// TwinCAT 3 PLC project Untitled1
// ProgramVersion: 3.1.4023.0
// libraries:
//   Tc2_EtherCAT, * (Beckhoff Automation GmbH)
//   Tc2_Standard, * (Beckhoff Automation GmbH)
//   Tc2_System, * (Beckhoff Automation GmbH)
//   Tc3_Module, * (Beckhoff Automation GmbH)
//   VisuDialogs, * (System)
// project tree:
//   DUTs/ DriveReference.TcDUT, Mat3.TcDUT, Motor.TcDUT, TorqueSensor.TcDUT, Vec3.TcDUT
//   / GlobalTextList.TcGTLO, PlcTask.TcTTO, 视图管理器.TcVMO (not stored)
//   GVLs/ GVL.TcGVL
//   POUs/controller/ IntegratedDrive.TcPOU, LegController.TcPOU
//   POUs/GaitPlanner/ BLegSlip.TcPOU, CurlingGait.TcPOU, CurlingGaitFromSlip.TcPOU, CurlingGaitFromStance.TcPOU, GaitPlanner.TcPOU, LiftBodyGait.TcPOU, RcToCurlingFromSlip.TcPOU, RcToSlipFromCurling.TcPOU, RcToStanceFromSlip.TcPOU, RecoverGait.TcPOU, SwingBodyGait.TcPOU, StaticWalkGait.TcPOU, TrotWalk.TcPOU, WalkSlopeGait.TcPOU
//   POUs/HardwareSetup/ MotorDriveSetup.TcPOU, SdoSetup.TcPOU
//   POUs/ MAIN.TcPOU, UIHandler.TcPOU
//   POUs/tools/ AngleCutFun.TcPOU, atan2Fun.TcPOU, CosGenerator.TcPOU, CubicSpline.TcPOU, ElipseInterpolation.TcPOU, GetPivot.TcPOU, HermitInterpolation.TcPOU, LowpassFilter.TcPOU, Min3Value.TcPOU, MinDistanceValue.TcPOU, RotM.TcPOU, SdoWrite.TcPOU
//   POUs/tools/VectorMath/ Atan2.TcPOU, Inv3.TcPOU, MatMulVec.TcPOU, MatTranspose.TcPOU, SetMat3.TcPOU, SetMat7_3.TcPOU, SetVec3.TcPOU, VecAdd.TcPOU, VecCross.TcPOU, VecMulNum.TcPOU, VecNeg.TcPOU, VecNorm.TcPOU, VecNormalize.TcPOU, VecSum.TcPOU
//   VISUs/ AxisControl.TcVIS, ForceControl.TcVIS, Monitor.TcVIS, RobotUI.TcVIS
// real-time tasks:
//   TASK PlcTask: cycle T#1ms, priority 20, ADS port 350
// I/O:
//   DEVICE Device 3 (EtherCAT), AmsNetId 10.0.0.119.4.1
//     Drive 1 (CiA402 Motor Control Device) [SOMANET CiA402 Drive]
//     Drive 2 (CiA402 Motor Control Device) [SOMANET CiA402 Drive]
//     Drive 3 (CiA402 Motor Control Device) [SOMANET CiA402 Drive]
//     Drive 4 (CiA402 Motor Control Device) [SOMANET CiA402 Drive]
//     Drive 5 (CiA402 Motor Control Device) [SOMANET CiA402 Drive]
//     Drive 6 (CiA402 Motor Control Device) [SOMANET CiA402 Drive]
//     Drive 7 (CiA402 Motor Control Device) [SOMANET CiA402 Drive]
//     Drive 8 (CiA402 Motor Control Device) [SOMANET CiA402 Drive]
//     Drive 9 (CiA402 Motor Control Device) [SOMANET CiA402 Drive]
//     Drive 10 (CiA402 Motor Control Device) [SOMANET CiA402 Drive]
//     Drive 11 (CiA402 Motor Control Device) [SOMANET CiA402 Drive]
//     Drive 12 (CiA402 Motor Control Device) [SOMANET CiA402 Drive]
//     Drive 13 (CiA402 Motor Control Device) [SOMANET CiA402 Drive]
//     Drive 14 (CiA402 Motor Control Device) [SOMANET CiA402 Drive]
//     Drive 15 (CiA402 Motor Control Device) [SOMANET CiA402 Drive]
//     Drive 16 (CiA402 Motor Control Device) [SOMANET CiA402 Drive]
//     Drive 17 (CiA402 Motor Control Device) [SOMANET CiA402 Drive]
//     Drive 18 (CiA402 Motor Control Device) [SOMANET CiA402 Drive]
//     Box 19 (TorqueGateway_IMU) [TorqueGateway_IMU]
//     Box 20 (TorqueGateway_IMU) [TorqueGateway_IMU]
//     Box 21 (TorqueGateway_IMU) [TorqueGateway_IMU]
//     Drive 22 (Diamond) [Diamond EtherCAT Drive]
//     Drive 23 (Diamond) [Diamond EtherCAT Drive]
//     Drive 24 (Diamond) [Diamond EtherCAT Drive]
// variable links:
//   Untitled1/Untitled1 Instance <-> Device 3 (EtherCAT)/Box 19 (TorqueGateway_IMU)
//     PlcTask Inputs/GVL.motorDrive[10].trqSensor.trqsensorValue <-> Axis3 process data mapping/ActTrq
//     PlcTask Inputs/GVL.motorDrive[11].trqSensor.trqsensorValue <-> Axis6 process data mapping/ActTrq
//     PlcTask Inputs/GVL.motorDrive[6].trqSensor.trqsensorValue <-> Axis1 process data mapping/ActTrq
//     PlcTask Inputs/GVL.motorDrive[7].trqSensor.trqsensorValue <-> Axis2 process data mapping/ActTrq
//     PlcTask Inputs/GVL.motorDrive[8].trqSensor.trqsensorValue <-> Axis4 process data mapping/ActTrq
//     PlcTask Inputs/GVL.motorDrive[9].trqSensor.trqsensorValue <-> Axis5 process data mapping/ActTrq
//     PlcTask Outputs/GVL.setTrqSensorZero[0] <-> Para process data mapping/Zero
//   Untitled1/Untitled1 Instance <-> Device 3 (EtherCAT)/Box 20 (TorqueGateway_IMU)
//     PlcTask Inputs/GVL.motorDrive[0].trqSensor.trqsensorValue <-> Axis5 process data mapping/ActTrq
//     PlcTask Inputs/GVL.motorDrive[15].trqSensor.trqsensorValue <-> Axis4 process data mapping/ActTrq
//     PlcTask Inputs/GVL.motorDrive[16].trqSensor.trqsensorValue <-> Axis1 process data mapping/ActTrq
//     PlcTask Inputs/GVL.motorDrive[17].trqSensor.trqsensorValue <-> Axis2 process data mapping/ActTrq
//     PlcTask Inputs/GVL.motorDrive[1].trqSensor.trqsensorValue <-> Axis6 process data mapping/ActTrq
//     PlcTask Inputs/GVL.motorDrive[2].trqSensor.trqsensorValue <-> Axis3 process data mapping/ActTrq
//     PlcTask Inputs/GVL.rpy_inpt[0] <-> POSE process data mapping/roll
//     PlcTask Inputs/GVL.rpy_inpt[1] <-> POSE process data mapping/pitch
//     PlcTask Inputs/GVL.rpy_inpt[2] <-> POSE process data mapping/yaw
//     PlcTask Outputs/GVL.setTrqSensorZero[1] <-> Para process data mapping/Zero
//   Untitled1/Untitled1 Instance <-> Device 3 (EtherCAT)/Box 21 (TorqueGateway_IMU)
//     PlcTask Inputs/GVL.motorDrive[12].trqSensor.trqsensorValue <-> Axis3 process data mapping/ActTrq
//     PlcTask Inputs/GVL.motorDrive[13].trqSensor.trqsensorValue <-> Axis6 process data mapping/ActTrq
//     PlcTask Inputs/GVL.motorDrive[14].trqSensor.trqsensorValue <-> Axis5 process data mapping/ActTrq
//     PlcTask Inputs/GVL.motorDrive[3].trqSensor.trqsensorValue <-> Axis4 process data mapping/ActTrq
//     PlcTask Inputs/GVL.motorDrive[4].trqSensor.trqsensorValue <-> Axis2 process data mapping/ActTrq
//     PlcTask Inputs/GVL.motorDrive[5].trqSensor.trqsensorValue <-> Axis1 process data mapping/ActTrq
//     PlcTask Outputs/GVL.setTrqSensorZero[2] <-> Para process data mapping/Zero
//   Untitled1/Untitled1 Instance <-> Device 3 (EtherCAT)/Drive 1 (CiA402 Motor Control Device)
//     PlcTask Inputs/GVL.motorDrive[11].motor.actualPos <-> TxPDO Mapping 1/Position actual value
//     PlcTask Inputs/GVL.motorDrive[11].motor.actualTrq <-> TxPDO Mapping 1/Torque actual value
//     PlcTask Inputs/GVL.motorDrive[11].motor.actualVel <-> TxPDO Mapping 1/Velocity actual value
//     PlcTask Inputs/GVL.motorDrive[11].motor.opModeDisp <-> TxPDO Mapping 1/Modes of operation display
//     PlcTask Inputs/GVL.motorDrive[11].motor.statusWord <-> TxPDO Mapping 1/Statusword
//     PlcTask Outputs/GVL.motorDrive[11].motor.ctrlWord <-> RxPDO Mapping 1/Controlword
//     PlcTask Outputs/GVL.motorDrive[11].motor.opMode <-> RxPDO Mapping 1/Modes of operation
//     PlcTask Outputs/GVL.motorDrive[11].motor.targetPos <-> RxPDO Mapping 1/Target position
//     PlcTask Outputs/GVL.motorDrive[11].motor.targetTrq <-> RxPDO Mapping 1/Target torque
//     PlcTask Outputs/GVL.motorDrive[11].motor.targetVel <-> RxPDO Mapping 1/Target velocity
//   Untitled1/Untitled1 Instance <-> Device 3 (EtherCAT)/Drive 10 (CiA402 Motor Control Device)
//     PlcTask Inputs/GVL.motorDrive[2].motor.actualPos <-> TxPDO Mapping 1/Position actual value
//     PlcTask Inputs/GVL.motorDrive[2].motor.actualTrq <-> TxPDO Mapping 1/Torque actual value
//     PlcTask Inputs/GVL.motorDrive[2].motor.actualVel <-> TxPDO Mapping 1/Velocity actual value
//     PlcTask Inputs/GVL.motorDrive[2].motor.opModeDisp <-> TxPDO Mapping 1/Modes of operation display
//     PlcTask Inputs/GVL.motorDrive[2].motor.statusWord <-> TxPDO Mapping 1/Statusword
//     PlcTask Outputs/GVL.motorDrive[2].motor.ctrlWord <-> RxPDO Mapping 1/Controlword
//     PlcTask Outputs/GVL.motorDrive[2].motor.opMode <-> RxPDO Mapping 1/Modes of operation
//     PlcTask Outputs/GVL.motorDrive[2].motor.targetPos <-> RxPDO Mapping 1/Target position
//     PlcTask Outputs/GVL.motorDrive[2].motor.targetTrq <-> RxPDO Mapping 1/Target torque
//     PlcTask Outputs/GVL.motorDrive[2].motor.targetVel <-> RxPDO Mapping 1/Target velocity
//   Untitled1/Untitled1 Instance <-> Device 3 (EtherCAT)/Drive 11 (CiA402 Motor Control Device)
//     PlcTask Inputs/GVL.motorDrive[1].motor.actualPos <-> TxPDO Mapping 1/Position actual value
//     PlcTask Inputs/GVL.motorDrive[1].motor.actualTrq <-> TxPDO Mapping 1/Torque actual value
//     PlcTask Inputs/GVL.motorDrive[1].motor.actualVel <-> TxPDO Mapping 1/Velocity actual value
//     PlcTask Inputs/GVL.motorDrive[1].motor.opModeDisp <-> TxPDO Mapping 1/Modes of operation display
//     PlcTask Inputs/GVL.motorDrive[1].motor.statusWord <-> TxPDO Mapping 1/Statusword
//     PlcTask Outputs/GVL.motorDrive[1].motor.ctrlWord <-> RxPDO Mapping 1/Controlword
//     PlcTask Outputs/GVL.motorDrive[1].motor.opMode <-> RxPDO Mapping 1/Modes of operation
//     PlcTask Outputs/GVL.motorDrive[1].motor.targetPos <-> RxPDO Mapping 1/Target position
//     PlcTask Outputs/GVL.motorDrive[1].motor.targetTrq <-> RxPDO Mapping 1/Target torque
//     PlcTask Outputs/GVL.motorDrive[1].motor.targetVel <-> RxPDO Mapping 1/Target velocity
//   Untitled1/Untitled1 Instance <-> Device 3 (EtherCAT)/Drive 12 (CiA402 Motor Control Device)
//     PlcTask Inputs/GVL.motorDrive[0].motor.actualPos <-> TxPDO Mapping 1/Position actual value
//     PlcTask Inputs/GVL.motorDrive[0].motor.actualTrq <-> TxPDO Mapping 1/Torque actual value
//     PlcTask Inputs/GVL.motorDrive[0].motor.actualVel <-> TxPDO Mapping 1/Velocity actual value
//     PlcTask Inputs/GVL.motorDrive[0].motor.opModeDisp <-> TxPDO Mapping 1/Modes of operation display
//     PlcTask Inputs/GVL.motorDrive[0].motor.statusWord <-> TxPDO Mapping 1/Statusword
//     PlcTask Outputs/GVL.motorDrive[0].motor.ctrlWord <-> RxPDO Mapping 1/Controlword
//     PlcTask Outputs/GVL.motorDrive[0].motor.opMode <-> RxPDO Mapping 1/Modes of operation
//     PlcTask Outputs/GVL.motorDrive[0].motor.targetPos <-> RxPDO Mapping 1/Target position
//     PlcTask Outputs/GVL.motorDrive[0].motor.targetTrq <-> RxPDO Mapping 1/Target torque
//     PlcTask Outputs/GVL.motorDrive[0].motor.targetVel <-> RxPDO Mapping 1/Target velocity
//   Untitled1/Untitled1 Instance <-> Device 3 (EtherCAT)/Drive 13 (CiA402 Motor Control Device)
//     PlcTask Inputs/GVL.motorDrive[5].motor.actualPos <-> TxPDO Mapping 1/Position actual value
//     PlcTask Inputs/GVL.motorDrive[5].motor.actualTrq <-> TxPDO Mapping 1/Torque actual value
//     PlcTask Inputs/GVL.motorDrive[5].motor.actualVel <-> TxPDO Mapping 1/Velocity actual value
//     PlcTask Inputs/GVL.motorDrive[5].motor.opModeDisp <-> TxPDO Mapping 1/Modes of operation display
//     PlcTask Inputs/GVL.motorDrive[5].motor.statusWord <-> TxPDO Mapping 1/Statusword
//     PlcTask Outputs/GVL.motorDrive[5].motor.ctrlWord <-> RxPDO Mapping 1/Controlword
//     PlcTask Outputs/GVL.motorDrive[5].motor.opMode <-> RxPDO Mapping 1/Modes of operation
//     PlcTask Outputs/GVL.motorDrive[5].motor.targetPos <-> RxPDO Mapping 1/Target position
//     PlcTask Outputs/GVL.motorDrive[5].motor.targetTrq <-> RxPDO Mapping 1/Target torque
//     PlcTask Outputs/GVL.motorDrive[5].motor.targetVel <-> RxPDO Mapping 1/Target velocity
//   Untitled1/Untitled1 Instance <-> Device 3 (EtherCAT)/Drive 14 (CiA402 Motor Control Device)
//     PlcTask Inputs/GVL.motorDrive[4].motor.actualPos <-> TxPDO Mapping 1/Position actual value
//     PlcTask Inputs/GVL.motorDrive[4].motor.actualTrq <-> TxPDO Mapping 1/Torque actual value
//     PlcTask Inputs/GVL.motorDrive[4].motor.actualVel <-> TxPDO Mapping 1/Velocity actual value
//     PlcTask Inputs/GVL.motorDrive[4].motor.opModeDisp <-> TxPDO Mapping 1/Modes of operation display
//     PlcTask Inputs/GVL.motorDrive[4].motor.statusWord <-> TxPDO Mapping 1/Statusword
//     PlcTask Outputs/GVL.motorDrive[4].motor.ctrlWord <-> RxPDO Mapping 1/Controlword
//     PlcTask Outputs/GVL.motorDrive[4].motor.opMode <-> RxPDO Mapping 1/Modes of operation
//     PlcTask Outputs/GVL.motorDrive[4].motor.targetPos <-> RxPDO Mapping 1/Target position
//     PlcTask Outputs/GVL.motorDrive[4].motor.targetTrq <-> RxPDO Mapping 1/Target torque
//     PlcTask Outputs/GVL.motorDrive[4].motor.targetVel <-> RxPDO Mapping 1/Target velocity
//   Untitled1/Untitled1 Instance <-> Device 3 (EtherCAT)/Drive 15 (CiA402 Motor Control Device)
//     PlcTask Inputs/GVL.motorDrive[3].motor.actualPos <-> TxPDO Mapping 1/Position actual value
//     PlcTask Inputs/GVL.motorDrive[3].motor.actualTrq <-> TxPDO Mapping 1/Torque actual value
//     PlcTask Inputs/GVL.motorDrive[3].motor.actualVel <-> TxPDO Mapping 1/Velocity actual value
//     PlcTask Inputs/GVL.motorDrive[3].motor.opModeDisp <-> TxPDO Mapping 1/Modes of operation display
//     PlcTask Inputs/GVL.motorDrive[3].motor.statusWord <-> TxPDO Mapping 1/Statusword
//     PlcTask Outputs/GVL.motorDrive[3].motor.ctrlWord <-> RxPDO Mapping 1/Controlword
//     PlcTask Outputs/GVL.motorDrive[3].motor.opMode <-> RxPDO Mapping 1/Modes of operation
//     PlcTask Outputs/GVL.motorDrive[3].motor.targetPos <-> RxPDO Mapping 1/Target position
//     PlcTask Outputs/GVL.motorDrive[3].motor.targetTrq <-> RxPDO Mapping 1/Target torque
//     PlcTask Outputs/GVL.motorDrive[3].motor.targetVel <-> RxPDO Mapping 1/Target velocity
//   Untitled1/Untitled1 Instance <-> Device 3 (EtherCAT)/Drive 16 (CiA402 Motor Control Device)
//     PlcTask Inputs/GVL.motorDrive[8].motor.actualPos <-> TxPDO Mapping 1/Position actual value
//     PlcTask Inputs/GVL.motorDrive[8].motor.actualTrq <-> TxPDO Mapping 1/Torque actual value
//     PlcTask Inputs/GVL.motorDrive[8].motor.actualVel <-> TxPDO Mapping 1/Velocity actual value
//     PlcTask Inputs/GVL.motorDrive[8].motor.opModeDisp <-> TxPDO Mapping 1/Modes of operation display
//     PlcTask Inputs/GVL.motorDrive[8].motor.statusWord <-> TxPDO Mapping 1/Statusword
//     PlcTask Outputs/GVL.motorDrive[8].motor.ctrlWord <-> RxPDO Mapping 1/Controlword
//     PlcTask Outputs/GVL.motorDrive[8].motor.opMode <-> RxPDO Mapping 1/Modes of operation
//     PlcTask Outputs/GVL.motorDrive[8].motor.targetPos <-> RxPDO Mapping 1/Target position
//     PlcTask Outputs/GVL.motorDrive[8].motor.targetTrq <-> RxPDO Mapping 1/Target torque
//     PlcTask Outputs/GVL.motorDrive[8].motor.targetVel <-> RxPDO Mapping 1/Target velocity
//   Untitled1/Untitled1 Instance <-> Device 3 (EtherCAT)/Drive 17 (CiA402 Motor Control Device)
//     PlcTask Inputs/GVL.motorDrive[7].motor.actualPos <-> TxPDO Mapping 1/Position actual value
//     PlcTask Inputs/GVL.motorDrive[7].motor.actualTrq <-> TxPDO Mapping 1/Torque actual value
//     PlcTask Inputs/GVL.motorDrive[7].motor.actualVel <-> TxPDO Mapping 1/Velocity actual value
//     PlcTask Inputs/GVL.motorDrive[7].motor.opModeDisp <-> TxPDO Mapping 1/Modes of operation display
//     PlcTask Inputs/GVL.motorDrive[7].motor.statusWord <-> TxPDO Mapping 1/Statusword
//     PlcTask Outputs/GVL.motorDrive[7].motor.ctrlWord <-> RxPDO Mapping 1/Controlword
//     PlcTask Outputs/GVL.motorDrive[7].motor.opMode <-> RxPDO Mapping 1/Modes of operation
//     PlcTask Outputs/GVL.motorDrive[7].motor.targetPos <-> RxPDO Mapping 1/Target position
//     PlcTask Outputs/GVL.motorDrive[7].motor.targetTrq <-> RxPDO Mapping 1/Target torque
//     PlcTask Outputs/GVL.motorDrive[7].motor.targetVel <-> RxPDO Mapping 1/Target velocity
//   Untitled1/Untitled1 Instance <-> Device 3 (EtherCAT)/Drive 18 (CiA402 Motor Control Device)
//     PlcTask Inputs/GVL.motorDrive[6].motor.actualPos <-> TxPDO Mapping 1/Position actual value
//     PlcTask Inputs/GVL.motorDrive[6].motor.actualTrq <-> TxPDO Mapping 1/Torque actual value
//     PlcTask Inputs/GVL.motorDrive[6].motor.actualVel <-> TxPDO Mapping 1/Velocity actual value
//     PlcTask Inputs/GVL.motorDrive[6].motor.opModeDisp <-> TxPDO Mapping 1/Modes of operation display
//     PlcTask Inputs/GVL.motorDrive[6].motor.statusWord <-> TxPDO Mapping 1/Statusword
//     PlcTask Outputs/GVL.motorDrive[6].motor.ctrlWord <-> RxPDO Mapping 1/Controlword
//     PlcTask Outputs/GVL.motorDrive[6].motor.opMode <-> RxPDO Mapping 1/Modes of operation
//     PlcTask Outputs/GVL.motorDrive[6].motor.targetPos <-> RxPDO Mapping 1/Target position
//     PlcTask Outputs/GVL.motorDrive[6].motor.targetTrq <-> RxPDO Mapping 1/Target torque
//     PlcTask Outputs/GVL.motorDrive[6].motor.targetVel <-> RxPDO Mapping 1/Target velocity
//   Untitled1/Untitled1 Instance <-> Device 3 (EtherCAT)/Drive 2 (CiA402 Motor Control Device)
//     PlcTask Inputs/GVL.motorDrive[10].motor.actualPos <-> TxPDO Mapping 1/Position actual value
//     PlcTask Inputs/GVL.motorDrive[10].motor.actualTrq <-> TxPDO Mapping 1/Torque actual value
//     PlcTask Inputs/GVL.motorDrive[10].motor.actualVel <-> TxPDO Mapping 1/Velocity actual value
//     PlcTask Inputs/GVL.motorDrive[10].motor.opModeDisp <-> TxPDO Mapping 1/Modes of operation display
//     PlcTask Inputs/GVL.motorDrive[10].motor.statusWord <-> TxPDO Mapping 1/Statusword
//     PlcTask Outputs/GVL.motorDrive[10].motor.ctrlWord <-> RxPDO Mapping 1/Controlword
//     PlcTask Outputs/GVL.motorDrive[10].motor.opMode <-> RxPDO Mapping 1/Modes of operation
//     PlcTask Outputs/GVL.motorDrive[10].motor.targetPos <-> RxPDO Mapping 1/Target position
//     PlcTask Outputs/GVL.motorDrive[10].motor.targetTrq <-> RxPDO Mapping 1/Target torque
//     PlcTask Outputs/GVL.motorDrive[10].motor.targetVel <-> RxPDO Mapping 1/Target velocity
//   Untitled1/Untitled1 Instance <-> Device 3 (EtherCAT)/Drive 22 (Diamond)
//     PlcTask Inputs/GVL.motorDrive[20].motor.actualPos <-> FeedBack process data mapping/Position actual value
//     PlcTask Inputs/GVL.motorDrive[20].motor.actualTrq <-> FeedBack process data mapping/Torque actual value
//     PlcTask Inputs/GVL.motorDrive[20].motor.actualVel <-> FeedBack process data mapping/Velocity actual value
//     PlcTask Inputs/GVL.motorDrive[20].motor.opModeDisp <-> FeedBack process data mapping/Modes of operation display
//     PlcTask Inputs/GVL.motorDrive[20].motor.statusWord <-> FeedBack process data mapping/Statusword
//     PlcTask Outputs/GVL.motorDrive[20].motor.ctrlWord <-> Reference process data mapping/Controlword
//     PlcTask Outputs/GVL.motorDrive[20].motor.opMode <-> Reference process data mapping/Modes of operation
//     PlcTask Outputs/GVL.motorDrive[20].motor.targetPos <-> Reference process data mapping/Target position
//     PlcTask Outputs/GVL.motorDrive[20].motor.targetTrq <-> Reference process data mapping/Target torque
//     PlcTask Outputs/GVL.motorDrive[20].motor.targetVel <-> Reference process data mapping/Target velocity
//   Untitled1/Untitled1 Instance <-> Device 3 (EtherCAT)/Drive 23 (Diamond)
//     PlcTask Inputs/GVL.motorDrive[19].motor.actualPos <-> FeedBack process data mapping/Position actual value
//     PlcTask Inputs/GVL.motorDrive[19].motor.actualTrq <-> FeedBack process data mapping/Torque actual value
//     PlcTask Inputs/GVL.motorDrive[19].motor.actualVel <-> FeedBack process data mapping/Velocity actual value
//     PlcTask Inputs/GVL.motorDrive[19].motor.opModeDisp <-> FeedBack process data mapping/Modes of operation display
//     PlcTask Inputs/GVL.motorDrive[19].motor.statusWord <-> FeedBack process data mapping/Statusword
//     PlcTask Outputs/GVL.motorDrive[19].motor.ctrlWord <-> Reference process data mapping/Controlword
//     PlcTask Outputs/GVL.motorDrive[19].motor.opMode <-> Reference process data mapping/Modes of operation
//     PlcTask Outputs/GVL.motorDrive[19].motor.targetPos <-> Reference process data mapping/Target position
//     PlcTask Outputs/GVL.motorDrive[19].motor.targetTrq <-> Reference process data mapping/Target torque
//     PlcTask Outputs/GVL.motorDrive[19].motor.targetVel <-> Reference process data mapping/Target velocity
//   Untitled1/Untitled1 Instance <-> Device 3 (EtherCAT)/Drive 24 (Diamond)
//     PlcTask Inputs/GVL.motorDrive[18].motor.actualPos <-> FeedBack process data mapping/Position actual value
//     PlcTask Inputs/GVL.motorDrive[18].motor.actualTrq <-> FeedBack process data mapping/Torque actual value
//     PlcTask Inputs/GVL.motorDrive[18].motor.actualVel <-> FeedBack process data mapping/Velocity actual value
//     PlcTask Inputs/GVL.motorDrive[18].motor.opModeDisp <-> FeedBack process data mapping/Modes of operation display
//     PlcTask Inputs/GVL.motorDrive[18].motor.statusWord <-> FeedBack process data mapping/Statusword
//     PlcTask Outputs/GVL.motorDrive[18].motor.ctrlWord <-> Reference process data mapping/Controlword
//     PlcTask Outputs/GVL.motorDrive[18].motor.opMode <-> Reference process data mapping/Modes of operation
//     PlcTask Outputs/GVL.motorDrive[18].motor.targetPos <-> Reference process data mapping/Target position
//     PlcTask Outputs/GVL.motorDrive[18].motor.targetTrq <-> Reference process data mapping/Target torque
//     PlcTask Outputs/GVL.motorDrive[18].motor.targetVel <-> Reference process data mapping/Target velocity
//   Untitled1/Untitled1 Instance <-> Device 3 (EtherCAT)/Drive 3 (CiA402 Motor Control Device)
//     PlcTask Inputs/GVL.motorDrive[9].motor.actualPos <-> TxPDO Mapping 1/Position actual value
//     PlcTask Inputs/GVL.motorDrive[9].motor.actualTrq <-> TxPDO Mapping 1/Torque actual value
//     PlcTask Inputs/GVL.motorDrive[9].motor.actualVel <-> TxPDO Mapping 1/Velocity actual value
//     PlcTask Inputs/GVL.motorDrive[9].motor.opModeDisp <-> TxPDO Mapping 1/Modes of operation display
//     PlcTask Inputs/GVL.motorDrive[9].motor.statusWord <-> TxPDO Mapping 1/Statusword
//     PlcTask Outputs/GVL.motorDrive[9].motor.ctrlWord <-> RxPDO Mapping 1/Controlword
//     PlcTask Outputs/GVL.motorDrive[9].motor.opMode <-> RxPDO Mapping 1/Modes of operation
//     PlcTask Outputs/GVL.motorDrive[9].motor.targetPos <-> RxPDO Mapping 1/Target position
//     PlcTask Outputs/GVL.motorDrive[9].motor.targetTrq <-> RxPDO Mapping 1/Target torque
//     PlcTask Outputs/GVL.motorDrive[9].motor.targetVel <-> RxPDO Mapping 1/Target velocity
//   Untitled1/Untitled1 Instance <-> Device 3 (EtherCAT)/Drive 4 (CiA402 Motor Control Device)
//     PlcTask Inputs/GVL.motorDrive[14].motor.actualPos <-> TxPDO Mapping 1/Position actual value
//     PlcTask Inputs/GVL.motorDrive[14].motor.actualTrq <-> TxPDO Mapping 1/Torque actual value
//     PlcTask Inputs/GVL.motorDrive[14].motor.actualVel <-> TxPDO Mapping 1/Velocity actual value
//     PlcTask Inputs/GVL.motorDrive[14].motor.opModeDisp <-> TxPDO Mapping 1/Modes of operation display
//     PlcTask Inputs/GVL.motorDrive[14].motor.statusWord <-> TxPDO Mapping 1/Statusword
//     PlcTask Outputs/GVL.motorDrive[14].motor.ctrlWord <-> RxPDO Mapping 1/Controlword
//     PlcTask Outputs/GVL.motorDrive[14].motor.opMode <-> RxPDO Mapping 1/Modes of operation
//     PlcTask Outputs/GVL.motorDrive[14].motor.targetPos <-> RxPDO Mapping 1/Target position
//     PlcTask Outputs/GVL.motorDrive[14].motor.targetTrq <-> RxPDO Mapping 1/Target torque
//     PlcTask Outputs/GVL.motorDrive[14].motor.targetVel <-> RxPDO Mapping 1/Target velocity
//   Untitled1/Untitled1 Instance <-> Device 3 (EtherCAT)/Drive 5 (CiA402 Motor Control Device)
//     PlcTask Inputs/GVL.motorDrive[13].motor.actualPos <-> TxPDO Mapping 1/Position actual value
//     PlcTask Inputs/GVL.motorDrive[13].motor.actualTrq <-> TxPDO Mapping 1/Torque actual value
//     PlcTask Inputs/GVL.motorDrive[13].motor.actualVel <-> TxPDO Mapping 1/Velocity actual value
//     PlcTask Inputs/GVL.motorDrive[13].motor.opModeDisp <-> TxPDO Mapping 1/Modes of operation display
//     PlcTask Inputs/GVL.motorDrive[13].motor.statusWord <-> TxPDO Mapping 1/Statusword
//     PlcTask Outputs/GVL.motorDrive[13].motor.ctrlWord <-> RxPDO Mapping 1/Controlword
//     PlcTask Outputs/GVL.motorDrive[13].motor.opMode <-> RxPDO Mapping 1/Modes of operation
//     PlcTask Outputs/GVL.motorDrive[13].motor.targetPos <-> RxPDO Mapping 1/Target position
//     PlcTask Outputs/GVL.motorDrive[13].motor.targetTrq <-> RxPDO Mapping 1/Target torque
//     PlcTask Outputs/GVL.motorDrive[13].motor.targetVel <-> RxPDO Mapping 1/Target velocity
//   Untitled1/Untitled1 Instance <-> Device 3 (EtherCAT)/Drive 6 (CiA402 Motor Control Device)
//     PlcTask Inputs/GVL.motorDrive[12].motor.actualPos <-> TxPDO Mapping 1/Position actual value
//     PlcTask Inputs/GVL.motorDrive[12].motor.actualTrq <-> TxPDO Mapping 1/Torque actual value
//     PlcTask Inputs/GVL.motorDrive[12].motor.actualVel <-> TxPDO Mapping 1/Velocity actual value
//     PlcTask Inputs/GVL.motorDrive[12].motor.opModeDisp <-> TxPDO Mapping 1/Modes of operation display
//     PlcTask Inputs/GVL.motorDrive[12].motor.statusWord <-> TxPDO Mapping 1/Statusword
//     PlcTask Outputs/GVL.motorDrive[12].motor.ctrlWord <-> RxPDO Mapping 1/Controlword
//     PlcTask Outputs/GVL.motorDrive[12].motor.opMode <-> RxPDO Mapping 1/Modes of operation
//     PlcTask Outputs/GVL.motorDrive[12].motor.targetPos <-> RxPDO Mapping 1/Target position
//     PlcTask Outputs/GVL.motorDrive[12].motor.targetTrq <-> RxPDO Mapping 1/Target torque
//     PlcTask Outputs/GVL.motorDrive[12].motor.targetVel <-> RxPDO Mapping 1/Target velocity
//   Untitled1/Untitled1 Instance <-> Device 3 (EtherCAT)/Drive 7 (CiA402 Motor Control Device)
//     PlcTask Inputs/GVL.motorDrive[17].motor.actualPos <-> TxPDO Mapping 1/Position actual value
//     PlcTask Inputs/GVL.motorDrive[17].motor.actualTrq <-> TxPDO Mapping 1/Torque actual value
//     PlcTask Inputs/GVL.motorDrive[17].motor.actualVel <-> TxPDO Mapping 1/Velocity actual value
//     PlcTask Inputs/GVL.motorDrive[17].motor.opModeDisp <-> TxPDO Mapping 1/Modes of operation display
//     PlcTask Inputs/GVL.motorDrive[17].motor.statusWord <-> TxPDO Mapping 1/Statusword
//     PlcTask Outputs/GVL.motorDrive[17].motor.ctrlWord <-> RxPDO Mapping 1/Controlword
//     PlcTask Outputs/GVL.motorDrive[17].motor.opMode <-> RxPDO Mapping 1/Modes of operation
//     PlcTask Outputs/GVL.motorDrive[17].motor.targetPos <-> RxPDO Mapping 1/Target position
//     PlcTask Outputs/GVL.motorDrive[17].motor.targetTrq <-> RxPDO Mapping 1/Target torque
//     PlcTask Outputs/GVL.motorDrive[17].motor.targetVel <-> RxPDO Mapping 1/Target velocity
//   Untitled1/Untitled1 Instance <-> Device 3 (EtherCAT)/Drive 8 (CiA402 Motor Control Device)
//     PlcTask Inputs/GVL.motorDrive[15].motor.actualPos <-> TxPDO Mapping 1/Position actual value
//     PlcTask Inputs/GVL.motorDrive[15].motor.actualTrq <-> TxPDO Mapping 1/Torque actual value
//     PlcTask Inputs/GVL.motorDrive[15].motor.actualVel <-> TxPDO Mapping 1/Velocity actual value
//     PlcTask Inputs/GVL.motorDrive[15].motor.opModeDisp <-> TxPDO Mapping 1/Modes of operation display
//     PlcTask Inputs/GVL.motorDrive[15].motor.statusWord <-> TxPDO Mapping 1/Statusword
//     PlcTask Outputs/GVL.motorDrive[15].motor.ctrlWord <-> RxPDO Mapping 1/Controlword
//     PlcTask Outputs/GVL.motorDrive[15].motor.opMode <-> RxPDO Mapping 1/Modes of operation
//     PlcTask Outputs/GVL.motorDrive[15].motor.targetPos <-> RxPDO Mapping 1/Target position
//     PlcTask Outputs/GVL.motorDrive[15].motor.targetTrq <-> RxPDO Mapping 1/Target torque
//     PlcTask Outputs/GVL.motorDrive[15].motor.targetVel <-> RxPDO Mapping 1/Target velocity
//   Untitled1/Untitled1 Instance <-> Device 3 (EtherCAT)/Drive 9 (CiA402 Motor Control Device)
//     PlcTask Inputs/GVL.motorDrive[16].motor.actualPos <-> TxPDO Mapping 1/Position actual value
//     PlcTask Inputs/GVL.motorDrive[16].motor.actualTrq <-> TxPDO Mapping 1/Torque actual value
//     PlcTask Inputs/GVL.motorDrive[16].motor.actualVel <-> TxPDO Mapping 1/Velocity actual value
//     PlcTask Inputs/GVL.motorDrive[16].motor.opModeDisp <-> TxPDO Mapping 1/Modes of operation display
//     PlcTask Inputs/GVL.motorDrive[16].motor.statusWord <-> TxPDO Mapping 1/Statusword
//     PlcTask Outputs/GVL.motorDrive[16].motor.ctrlWord <-> RxPDO Mapping 1/Controlword
//     PlcTask Outputs/GVL.motorDrive[16].motor.opMode <-> RxPDO Mapping 1/Modes of operation
//     PlcTask Outputs/GVL.motorDrive[16].motor.targetPos <-> RxPDO Mapping 1/Target position
//     PlcTask Outputs/GVL.motorDrive[16].motor.targetTrq <-> RxPDO Mapping 1/Target torque
//     PlcTask Outputs/GVL.motorDrive[16].motor.targetVel <-> RxPDO Mapping 1/Target velocity

CONFIGURATION Untitled1
    RESOURCE PLC ON TwinCAT3
        TASK PlcTask(INTERVAL := T#1ms, PRIORITY := 20);
        PROGRAM MAIN WITH PlcTask : MAIN;
    END_RESOURCE
END_CONFIGURATION

// ---- DUTs/DriveReference.TcDUT
TYPE DriveReference :
STRUCT
	drive : REFERENCE TO IntegratedDrive;
END_STRUCT
END_TYPE

// ---- DUTs/Mat3.TcDUT
TYPE Mat3 :
STRUCT
	data : ARRAY[0..2, 0..2] OF LREAL;
END_STRUCT
END_TYPE

// ---- DUTs/Motor.TcDUT
TYPE Motor :
STRUCT
	statusWord AT%I*: UINT;
	opModeDisp AT%I*: SINT;
	actualPos  AT%I*: DINT;  
	actualVel  AT%I*: DINT;  
	actualTrq  AT%I*: INT; 
	digInputs  AT%I*: DINT;
	
	ctrlWord   AT%Q*: UINT;
	opMode     AT%Q*: USINT;
    targetPos  AT%Q*: DINT   :=0;  
	targetVel  AT%Q*: DINT   :=0;
	targetTrq  AT%Q*: INT    :=0;
	maxTrq     AT%Q*: INT    :=2000;
END_STRUCT
END_TYPE

// ---- DUTs/TorqueSensor.TcDUT
TYPE TorqueSensor :
STRUCT
	trqsensorValue AT%I* : REAL; 
	targetTrqValue AT%I* : REAL;
    
	actPos         AT%Q* : REAL;
	actVel         AT%Q* : REAL;
	TgtPos         AT%Q* : REAL;
	TgtVel         AT%Q* : REAL;
	TrqOff         AT%Q* : REAL;
	SetCtrlPrm     AT%Q* : USINT; 
	reqReset      : usint := 0;
	
	signalPosSlope: LREAL := 35;
	signalNegSlope: LREAL := 35;
END_STRUCT
END_TYPE

// ---- DUTs/Vec3.TcDUT
TYPE Vec3 :
STRUCT
	data : ARRAY[0..2] OF LREAL;
END_STRUCT
END_TYPE

// ---- GVLs/GVL.TcGVL
{attribute 'qualified_only'}
VAR_GLOBAL
	
	
	(*yk 适应*)
	motor_count :  INT :=20;
	
	
	(* system parameters *)
	sampleRate              : DINT := 1000;
	//count2radianRatio  : LREAL := 5.9921124526782860535862796464529E-6;  // 2*pi/1048576
	count2radianRatio  : ARRAY[0..20] OF LREAL := [2*pi/1048576.0,2*pi/1048576.0,2*pi/1048576.0,
                                                   2*pi/1048576.0,2*pi/1048576.0,2*pi/1048576.0,
                                                   2*pi/1048576.0,2*pi/1048576.0,2*pi/1048576.0,
                                                   2*pi/1048576.0,2*pi/1048576.0,2*pi/1048576.0,
                                                   2*pi/1048576.0,2*pi/1048576.0,2*pi/1048576.0,
                                                   2*pi/1048576.0,2*pi/1048576.0,2*pi/1048576.0,
                                                   2*pi/4096.0/9.0,2*pi/4096.0/9.0,2*pi/4096.0/9.0];	
	(* hardware instances *)
	motorDrive              : ARRAY[0..20] OF IntegratedDrive;
	setTrqSensorZero AT%Q*  : ARRAY[0..2]  OF USINT;
	setCtrlZero      AT%Q*  : ARRAY[0..2]  OF USINT;
	
	(* sdo defs *)
	sdoSetup                : SdoSetup;
	sdoWriteOnce            : SdoWrite;
	
	(* IMU readings *)
	IMUDATA : ARRAY[1..6] OF LREAL;
	roll, pitch, yaw        : LREAL;
	accx, accy, accz        : LREAL;
	(* RPY angle aligned to model axis *)
	rpy_model               : ARRAY[0..2] OF LREAL;
	rpy_inpt 		   AT%I*: ARRAY[0..2] OF REAL;
	
	(* motor init parameters*)
	motorDirs        : ARRAY[0..20] OF INT := [1, -1, 1, 
                                               1, 1, 1,
                                               1, 1, 1,
                                               -1, -1, 1,
											   -1, -1, 1,
											   -1, 1, 1,-1,-1,1];//curling2
	(*trqSensorDirs    : ARRAY[0..19] OF INT := [1, -1, 1, 
                                               1, 1, 1,
                                               1, 1, 1,
                                               -1, -1, 1,
											   -1, -1, 1,
 											   -1, 1, 1,1,1];*)
	trqSensorDirs    : ARRAY[0..20] OF INT := [1, -1, 1, 
                                               1, 1, 1,
                                               1, 1, 1,
                                               -1, -1, 1,
											   -1, -1, 1,
 											   -1, 1, 1,-1,-1,-1];											   
											   
	// yk 按照小腿、大腿、侧摆角给出
	(*posHomeOffsets   : ARRAY[0..19] OF LREAL:= [5.497-pi, 3.9269, 0, 
                                                3.9269-pi, 5.497, 0,
                                                3.9269-pi, 5.497, -pi/2, 
                                                3.9269-pi, 5.497, pi/2,
							 					3.9269-pi, 5.497, 0, 
                                                5.497-pi, 3.9269, 0,0,0];//home position in model*)
	(*posHomeOffsets   : ARRAY[0..20] OF LREAL:= [316.8582*pi/180+0.0844, 103.423*pi/180+0.0636, 0*pi/180-0.012, 
                                                109.534*pi/180+0.0052, 350.2283*pi/180-0.042, 90*pi/180-0.018,
                                                102.1787*pi/180+0.0218, 322.4662*pi/180-0.0564, 90*pi/180-0.035, 
                                                102.1787*pi/180+0.0018, 322.4662*pi/180-0.0184, -90*pi/180+0.072,
							 					109.534*pi/180+0.0392, 350.2283*pi/180-0.061, -90*pi/180+0.032, 
                                                316.8582*pi/180+0.0954, 103.423*pi/180+0.0646,  0*180/pi-0,
												0,0,0*pi/180];//home position in model obtained by calibration board	*)
	posHomeOffsets   : ARRAY[0..20] OF LREAL:= [316.8582*pi/180+0.0844, 103.423*pi/180+0.0636, 0*pi/180-0.012, 
                                                109.534*pi/180+0.0052, 350.2283*pi/180-0.042, 90*pi/180-0.018,
                                                102.1787*pi/180+0.0218, 322.4662*pi/180-0.0564, 90*pi/180-0.035, 
                                                102.1787*pi/180+0.0018, 322.4662*pi/180-0.0184, -90*pi/180+0.072,
							 					109.534*pi/180+0.0392, 350.2283*pi/180-0.061, -90*pi/180+0.032, 
                                                316.8582*pi/180+0.0954, 103.423*pi/180+0.0646,  0*180/pi-0,
												0,0,0*pi/180];//home position in model obtained by calibration board											
														
	(*motorActualHomePosIncrement:ARRAY[0..20] OF DINT:= [-391364,-52566,310018,
														 -412094,-268692,-444796,	
														 -432711,-284347,268081,
														 343587,27385,507790,
														 -90255,27553,164936,
														 -124974,-465365,520356,
														 0,0,0];//increment at home position in model obtained by calibration board 20220104*)	
	motorActualHomePosIncrement:ARRAY[0..20] OF DINT:= [-391364,-52566,-281217,
														 -412094,-268692,-444796,	
														 -432711,-284347,268081,
														 343587,27385,507790,
														 -90255,27553,164936,
														 -124974,-465365,263290,
														 0,0,0];//increment at home position in model obtained by calibration board 20220104												 
														 
	signalPosSlopes   : ARRAY[0..20] OF LREAL := [65, 65, 65, 
                                               65, 65, 65,
                                               65, 65, 65,
                                               65, 65, 65,
											   65, 65, 65,
											   65, 65, 65,1,1,1];
	signalNegSlopes   : ARRAY[0..20] OF LREAL := [65, 65, 65, 
                                               65, 65, 65,
                                               65, 65, 65,
                                               65, 65, 65,
											   65, 65, 65,
											   65, 65, 65,1,1,1];
	homingVels       : ARRAY[0..20] OF LREAL:= [0.01, 0.01,  0.01, 
                                               0.01, 0.01,  0.01,
                                               0.01, 0.01,  0.01, 
                                               0.01, 0.01,  0.01,
											   0.01, 0.01,  0.01, 
                                               0.01, 0.01,  0.01,0,0,0.01];
	AbsMoveTgtPos  :	ARRAY[0..20] OF LREAL :=[0, 0, 0,
                                                          0, 0, 0,
														  0, 0, 0,
														  0, 0, 0,
														  0, 0, 0,
														  0, 0, 0,
			                                              0, 0, 0];												   
	redcClbConsts    : ARRAY[0..20] OF LREAL:= [0.01, 0.01, 0.01, 
                                                0.01, 0.01, 0.01,
                                                0.01, 0.01, 0.01, 
                                                0.01, 0.01, 0.01,
                                                0.01, 0.01, 0.01, 
                                                0.01, 0.01, 0.01,0,0,0];
	KPP_init    	 : ARRAY[0..20] OF LREAL:= [1250, 1250, 1250, 
                                                1250, 1250, 1250,
                                                1250, 1250, 1250, 
                                                1250, 1250, 1250,
                                                1250, 1250, 1250, 
                                                1250, 1250, 1250,0,0,0];	
	(*KPP_init    	 : ARRAY[0..20] OF LREAL:= [1000, 1000, 1000, 
                                                1000, 1000, 1000,
                                                1000, 1000, 1000, 
                                                1000, 1000, 1000,
                                                1000, 1000, 1000, 
                                                1000, 1000, 1000,0,0,0];	*)	
	KPD_init    	 : ARRAY[0..20] OF LREAL:= [25, 25, 25, 
                                                25, 25, 25,
                                                25, 25, 25, 
                                                25, 25, 25,
                                                25, 25, 25, 
                                                25, 25, 25,0,0,0];									
	(*KPD_init    	 : ARRAY[0..20] OF LREAL:= [10, 10, 10, 
                                                10, 10, 10,
                                                10, 10, 10, 
                                                10, 10, 10,
                                                10, 10, 10, 
                                                10, 10, 10,0,0,0];*)
	KFP_init    	 : ARRAY[0..20] OF LREAL:= [0.5, 0.5, 0.5, 
                                                0.5, 0.5, 0.5,
                                                0.5, 0.5, 0.5, 
                                                0.5, 0.5, 0.5,
                                                0.5, 0.5, 0.5, 
                                                0.5, 0.5, 0.5,0,0,0];
	KFI_init    	 : ARRAY[0..20] OF LREAL:= [0.75, 0.75, 0.75, 
                                                0.75, 0.75, 0.75,
                                                0.75, 0.75, 0.75, 
                                                0.75, 0.75, 0.75,
                                                0.75, 0.75, 0.75, 
                                                0.75, 0.75, 0.75,0,0,0];


													
												
	//yk 小腿、大腿、侧摆顺序给出，	电机实际角度值，只有运动学上角度才使用小腿角度+pi，			
	trqCtrlUpperAngs : ARRAY[0..20] OF LREAL:= [360, 360, 180, 
                                                360, 360, 180,
                                                360, 360, 180, 
                                                360, 360, 180,
                                                360, 360, 180, 
                                                360, 360, 180,180,180,360];
	trqCtrlLowerAngs : ARRAY[0..20] OF LREAL:= [0, 0, -180, 
                                                0, 0, -180,
                                                0, 0, -180, 
                                                0, 0, -180,
                                                0, 0, -180, 
                                                0, 0, -180,-180,-180,0];
	normalAngles   : ARRAY[0..20] OF LREAL:= [5.497, 3.9269, 0, 
                                              3.9269, 5.497, 0,
                                              3.9269, 5.497, 0, 
                                              3.9269, 5.497, 0,
                                              3.9269, 5.497, 0, 
                                              5.497, 3.9269, 0,0,0,0];// yk 小腿电机角度一定要小于大腿电机角度，才能保证平行四边形腿结构
	(* Visulization linked variables *)
	uiHandler             : UIHandler;
	
	(* axis command *)
	opModeCmd: ARRAY[0..20] OF USINT;
	enableCmd: ARRAY[0..20] OF BOOL;
	
	(* leg physical parameter *)
	ShankLength : ARRAY[0..5] OF LREAL:=[0.5,0.28,0.28,0.28,0.28,0.5];//RB,RM,RF,LF,LM,LB
	ThighLength : ARRAY[0..5] OF LREAL:=[0.5,0.3,0.3,0.3,0.3,0.5];//RB,RM,RF,LF,LM,LB
	
	(* model *)
	legCtrl               : ARRAY[0..5] OF LegController;
	sagPlaneOffset	  :ARRAY[0..5] OF LREAL:=[0,0.1246,0.1246,-0.1246,-0.1246,0];
	
	tipActualPos          : ARRAY[0..5,0..2] OF LREAL := [0, 0, 0,
                                                          0, 0, 0,
														  0, 0, 0,
														  0, 0, 0,
														  0, 0, 0,
														  0, 0, 0];
    tipActualVel          : ARRAY[0..5,0..2] OF LREAL := [0, 0, 0,
                                                          0, 0, 0,
														  0, 0, 0,
														  0, 0, 0,
														  0, 0, 0,
														  0, 0, 0];
    tipActualFce          : ARRAY[0..5,0..2] OF LREAL := [0, 0, 0,
                                                          0, 0, 0,
														  0, 0, 0,
														  0, 0, 0,
														  0, 0, 0,
														  0, 0, 0];
	// joint pos, vel and fce after hardware-model mapping
	jntActualPos          : ARRAY[0..5,0..2] OF LREAL := [0, 0, 0,
                                                          0, 0, 0,
														  0, 0, 0,
														  0, 0, 0,
														  0, 0, 0,
														  0, 0, 0];
    jntActualVel          : ARRAY[0..5,0..2] OF LREAL := [0, 0, 0,
                                                          0, 0, 0,
														  0, 0, 0,
														  0, 0, 0,
														  0, 0, 0,
														  0, 0, 0];
    jntActualFce          : ARRAY[0..5,0..2] OF LREAL := [0, 0, 0,
                                                          0, 0, 0,
														  0, 0, 0,
														  0, 0, 0,
														  0, 0, 0,
														  0, 0, 0];
	// yk 参考位置和速度按照单腿运动学侧摆、大腿、小腿（+pi）给出
	jntRefPos             : ARRAY[0..5,0..2] OF LREAL;
	jntRefVel             : ARRAY[0..5,0..2] OF LREAL;
	lastjntRefPos         : ARRAY[0..5,0..2] OF LREAL:=[0,0,0,
														0,0,0,
														0,0,0,
														0,0,0,
														0,0,0,
														0,0,0];
	jntRefVelDif          : ARRAY[0..5,0..2] OF LREAL;
	jntRefFce             : ARRAY[0..5,0..2] OF LREAL;
	jntLastRefPos         : ARRAY[0..5,0..2] OF LREAL;
	
	jntRefPosTuning       : ARRAY[0..5,0..2] OF LREAL;
	jntRefVelTuning       : ARRAY[0..5,0..2] OF LREAL;
	jntRefFceTuning       : ARRAY[0..5,0..2] OF LREAL;
	
	jntRefPosLastPlanning:ARRAY[0..5,0..2] OF LREAL;
	
	(*jntRefPosLastPlanningFirstRc:ARRAY[0..5,0..2] OF LREAL:=[0,188.4468*pi/180,322.1064*pi/180,
											 0,312.3065*pi/180,(219.5084-312.3065)*pi/180,	
											 0,312.3065*pi/180,(219.5084-312.3065)*pi/180,
											 0,312.3065*pi/180,(219.5084-312.3065)*pi/180,
									         0,312.3065*pi/180,(219.5084-312.3065)*pi/180,
											 0,188.4468*pi/180,322.1064*pi/180];*)
											 
	(*jntRefPosLastPlanningFirstRc:ARRAY[0..5,0..2] OF LREAL:=[0,194.9664*pi/180,320.003*pi/180,
											 0,302.7132*pi/180,(230.9946-302.7132)*pi/180,	
											 0,302.7132*pi/180,(230.9946-302.7132)*pi/180,
											 0,302.7132*pi/180,(230.9946-302.7132)*pi/180,
									         0,302.7132*pi/180,(230.9946-302.7132)*pi/180,
											 0,194.9664*pi/180,320.003*pi/180];	*)

	jntRefPosLastPlanningFirstRc:ARRAY[0..5,0..2] OF LREAL:=[0,156.4222*pi/180,269.8005*pi/180,
											 0,320.9331*pi/180,(208.0880-320.9331)*pi/180,	
											 0,187.8384*pi/180,(269.4264-187.8384)*pi/180,
											 0,187.8384*pi/180,(269.4264-187.8384)*pi/180,
									         0,320.9331*pi/180,(208.0880-320.9331)*pi/180,
											 0,156.4222*pi/180,269.8005*pi/180];										 
	
	(* axis control *)
	enablebuttonText      : ARRAY[0..20] OF STRING(20);
	enableButton          : ARRAY[0..20] OF BOOL;//赋值给enableCmd,gvl.motorDrive[i].DriverControl(gvl.opModeCmd[i], gvl.enableCmd[i])控制电机
	startHomeButton       : ARRAY[0..20] OF BOOL;//单轴和批量都可以赋值，批量赋值后需要进入单轴控制函数执行走home
	setInitPositionButton : ARRAY[0..20] OF BOOL;//单轴和批量都可以赋值，批量赋值后需要进入单轴控制函数执行走设置初始值，调用驱动器驱动函数设置当前home值进入驱动器
	jogButton             : ARRAY[0..20] OF BOOL;
	jogStopButton         : ARRAY[0..20] OF BOOL; 
	jogVelocity           : ARRAY[0..20] OF LREAL;
	AbsMoveButton		  : ARRAY[0..20] OF BOOL;
	AbsMoveStopButton	  : ARRAY[0..20] OF BOOL;
	
	setTSRZeroButton      : BOOL  := FALSE;
	groupSelector         : UINT  := 0;//单选对应数组号，为其值
	enableGroupButton     : BOOL  := FALSE;
	disableGroupButton    : BOOL  := FALSE;
	homeGroupButton       : BOOL  := FALSE;
	setPosGroupButton     : BOOL  := FALSE;
	jogGroupButton        : BOOL  := FALSE;
	jogStopGroupButton    : BOOL  := FALSE;
    //jogGroupVelocity      : DINT  := -2000;
	jogGroupVelocity      : lreal  := 0.01;
	
	setGroupImpedButton   : BOOL  := FALSE;
	useHardImpedButton    : BOOL  := FALSE;
	useSoftImpedButton    : BOOL  := FALSE;
	kpGroup               : LREAL := 220;
	kdGroup               : LREAL := 30;
	kpTrqGroup            : LREAL := 0.5;
	kiTrqGroup            : LREAL := 0.75;
	
	activeAxisList        : ARRAY[0..9] OF ARRAY[0..17] OF USINT := 
                              [[1,1,1,1,1,1,1,1,1,1,1,1,1,1,1,1,1,1],
                               [1,0,0,1,0,0,1,0,0,1,0,0,1,0,0,1,0,0],
                               [0,1,0,0,1,0,0,1,0,0,1,0,0,1,0,0,1,0],
                               [0,0,1,0,0,1,0,0,1,0,0,1,0,0,1,0,0,1],
                               [1,1,1,0,0,0,0,0,0,0,0,0,0,0,0,0,0,0],
                               [0,0,0,1,1,1,0,0,0,0,0,0,0,0,0,0,0,0],
                               [0,0,0,0,0,0,1,1,1,0,0,0,0,0,0,0,0,0],
                               [0,0,0,0,0,0,0,0,0,1,1,1,0,0,0,0,0,0],
                               [0,0,0,0,0,0,0,0,0,0,0,0,1,1,1,0,0,0],
                               [0,0,0,0,0,0,0,0,0,0,0,0,0,0,0,1,1,1]]; //yk 控制一起走home的驱动器号
	
	axisForceCtrlButton   : ARRAY[0..17] OF BOOL;//控制力控开始结束
	axisForceCtrlModeInd  : ARRAY[0..17] OF BOOL;//显示是否处于力控状态
	forceCtrlGroupButton     : BOOL := FALSE;//批量控制进入力控模式
	forceCtrlGroupOffButton  : BOOL := FALSE;//批量停止进入力控模式

	(* gait control *)
	startGaitButton: BOOL   := FALSE;
	isInGaitMode  :  BOOL   := FALSE;
	isFinished    :  BOOL   := FALSE;
	gaitPlanner   :  GaitPlanner;
	gaitId        :  UINT   := 0;
	gaitNameLists :  ARRAY[0..11] OF WSTRING(20) := ["Recovery", "Walk_static", "LiftBody", "Swing","CurlingFrStand","CurlingFrSlip","RcToSlipFrCurl","RcToCurFrSlip","RcToStandFrSlip","BLegSlip","TrotWalk","WalkSlope"];
	
	RcGaitId:UINT:=0;
	RcGaitNameLists:ARRAY[0..1] OF WSTRING(20):=["RcWalk","RcCurling"];
	
	(* measurement *)
	trqReadings           : ARRAY[0..17] OF LREAL;
	trqOutputs            : ARRAY[0..17] OF LREAL;
	trqOutputs2           : ARRAY[0..17] OF LREAL;
	jntActCurrentMea      : ARRAY[0..17] OF INT;
	jntActualPosMea       : ARRAY[0..3,0..2] OF REAL := [0, 0, 0,
                                                          0, 0, 0,
														  0, 0, 0,
														  0, 0, 0];

    jntActualFceMea       : ARRAY[0..3,0..2] OF REAL := [0, 0, 0,
                                                          0, 0, 0,
														  0, 0, 0,
														  0, 0, 0];
	
	jntRefPosMea          : ARRAY[0..3,0..2] OF REAL;
	jntRefFceMea          : ARRAY[0..3,0..2] OF REAL;
	
	(* global stop to shutdown all drives *)
	emergencyStop: BOOL := FALSE;//针对力控
	emergencyStopCount: INT := 0;
	
	(* trq sensor board *)
	useParamIndex: USINT;
	requireSet: BOOL := FALSE;
	raiseEdgeCount: INT := -1;
	setBit: USINT;
	
	walk_threshold_value:LREAL:=0.3;
    lift_threshold_value:LREAL:=0.3;
	swing_threshold_value:LREAL:=0.3;
	curling_threshold_value:lreal:=0.3;

	//Rc gait
	setRcRefAngButton:BOOL:=FALSE;
	
	//curling
	taskChooseId:UINT:=0;
	taskChooseList:array [0..1] of wstring(20):=["击打","进营"];
	adjust_angle_degree:LREAL:=0;//degree
	target_vel:LREAL:=2;//m/s
	stone_rot_vel:LREAL:=-60;//rpm
	PushVelocityIn:LREAL:=2.3;
	BPA_adjust_angle_degree:LREAL:=0;//degree
	BPA_adjust_x:LREAL:=-0.1;
	BPA_adjust_y:LREAL:=0;
	BLPA_adjust_distance_desire:ARRAY[0..1,0..2] OF LREAL:=[0,0,0,
															0,0,0];//[0,-0.01,0,0,0.01,0]																												
	curlingPushModel        :  UINT   := 0;
	curlingPushModelList :  ARRAY[0..1] OF WSTRING(20) := ["Push", "noPush"];
	PushFinishDurationTimeIn:LREAL:=1;
	slideTimeIn:LREAL:=0.3;
	ArmRetractControl:BOOL:=FALSE;
	AC_AngleDegIn:LREAL:=-40;
	
	gripBallThighTargetAngle:LREAL:=167.5;
	gripBallShankTargetAngle:LREAL:=171;
	
	//init value
	adjust_angle_degree_init:LREAL:=0;//degree
	target_vel_init:LREAL:=2;//m/s
	stone_rot_vel_init:LREAL:=-60;//rpm
	PushVelocityIn_init:LREAL:=2.3;
	BPA_adjust_angle_degree_init:LREAL:=0;//degree
	BPA_adjust_x_init:LREAL:=-0.1;
	BPA_adjust_y_init:LREAL:=0;
	BLPA_adjust_distance_desire_init:ARRAY[0..1,0..2] OF LREAL:=[0,0,0,
															0,0,0];	
	curlingPushModel_init        :  UINT   := 0;	
	PushFinishDurationTimeIn_init:LREAL:=1;
	slideTimeIn_init:LREAL:=0.3;
	ArmRetractControl_init:BOOL:=FALSE;
	AC_AngleDegIn_init:LREAL:=-40;	

	//BLegSlip
	BLegSlip_trot_vel_desire:LREAL:=0;
	BLegSlip_side_vel_desire:LREAL:=0;
	BLegSlip_turn_rate_desire:LREAL:=0;
	BLegSlip_step:ARRAY [0..2] OF LREAL:=[0.05,0.05,0.05];
	
	//TrotWalk
	TrotWalk_trot_vel_desire:LREAL:=0;
	TrotWalk_side_vel_desire:LREAL:=0;
	TrotWalk_turn_rate_desire:LREAL:=0;
	TrotWalk_step:ARRAY [0..2] OF LREAL:=[0.15,0.15,0.15];	
	period_desire:LREAL:=1.4;
	duty_desire:LREAL:=0.5;
	step_height_desire:LREAL:=0.06;
	
	//liftbody
	RestButton:BOOL:=FALSE;
	WorkButton:BOOL:=FALSE;
	ReduceDistance:LREAL:=-0.08;
	IsRest:BOOL:=FALSE;
	IsRcCurling:BOOL:=FALSE;
	IsPreLiftBody:BOOL:=FALSE;
	IsLiftBody:BOOL:=FALSE;
	RcEndFlagLast:BOOL:=FALSE;
	RcStartFlag:BOOL:=FALSE;
	RcEndFlag:BOOL:=FALSE;
	EnterPreLiftBodyCount:UDINT:=0;
	LiftBodyStartFlag:BOOL:=FALSE;
	LiftBodyEndFlag:BOOL:=FALSE;
	LiftBodyEndFlagLast:BOOL:=FALSE;
	
	IsWork:BOOL:=FALSE;
	
END_VAR

// ---- POUs/MAIN.TcPOU
PROGRAM MAIN
VAR
	i : UINT;
	j : UINT;
	count : UDINT := 0;

	tipPos, tipVel, tipFce : ARRAY[0..2] OF LREAL;
END_VAR

//////////////////////////////////////////////////////
//                                                  //
// Initialization                                   //
//                                                  //
//////////////////////////////////////////////////////
IF count = 0 THEN
	// init visulization parameters
	gvl.uiHandler.Initialize();
	// init message
	
	// init device address
	// with sdo settings
	gvl.sdoSetup.SetSlaveAddr();//yk需要根据控制器网址设置地址
	
	
	// init axes configuration
	// Note: Some parameters are downloaded to sdo
	// thus not all of these parameters are actually used
	FOR i := 0 TO 20 DO
		gvl.motorDrive[i].InitParam(
			// actual motor direction with regards to the model definition, -1 or +1
			motorDirIn      := gvl.motorDirs[i],
			// actual trq sensor direction wrt the model defintion, -1 or +1 
			trqSensorDirIn  := gvl.trqSensorDirs[i],
			// position offset at home ,need calibrate
			posHomeOffsetIn := gvl.posHomeOffsets[i],
			// signal positive slope of the torque sensor raw output to Nm
			signalPosSlope  := gvl.signalPosSlopes[i],
			// signal negative slope of the torque sensor raw output to Nm
			signalNegSlope  := gvl.signalNegSlopes[i],
			// home velocity
			homingVel       := gvl.homingVels[i],
			// constant of the coloumb friction, yk阻抗控制的是减速机输出扭矩，默认0.01Nm是作用在电机轴上。
			redcClbConst    := gvl.redcClbConsts[i] * 50,
			// trq ctrl upper angle, if the motor runs over this angle, it will be powered off 
			trqCtrlUpperAng := gvl.trqCtrlUpperAngs[i]/180.0*pi,
			// trq ctrl lower angle, if the motor runs over this angle, it will be powered off 
			trqCtrlLowerAng := gvl.trqCtrlLowerAngs[i]/180.0*Pi,
			// trq ctrl normal angle//电机实际值
			tgtAngleIn      := gvl.normalAngles[i]/180.0*pi,
			motorActualHomePosIncrementIn:=gvl.motorActualHomePosIncrement[i],
			indexIn:=i,
			kVirtualIn:=gvl.KPP_init[i],
			bVirtualIn:=gvl.KPD_init[i],
			kpTrqLoopIn:=gvl.KFP_init[i],
			kiTrqLoopIn:=gvl.KFI_init[i],
			count2radianRatioIn:=gvl.count2radianRatio[i]
		);
	END_FOR
	
	// configure leg parameters to leg controller
	FOR i := 0 TO 5 DO
		gvl.LegCtrl[i].InitParam(
			// leg id
			id := i,
			// length of shank link
			ShankLengthIn := GVL.ShankLength[i],
			// length of thigh link
			ThighLengthIn := GVL.ThighLength[i],
			// sagital plane offset
			sagPlaneOffsetIn:=gvl.sagPlaneOffset[i]);
	END_FOR
	
	// set RC reference
	gvl.jntRefPosLastPlanning:=gvl.jntRefPosLastPlanningFirstRc;
	
END_IF

//////////////////////////////////////////////////////
//                                                  //
// Cyclic control                                   //
//                                                  //
//////////////////////////////////////////////////////

// add count 
count := count + 1;

// write sdos configurations to devices 
// this command will last until the sdo writing ops finished 
 gvl.sdoSetup.InitSdoConfig();//设定走home模式和home对应0，所以角度换算时需要加入home对应实际运动学值,设置扭矩传感器可以删除

// update device feedbacks
FOR i := 0 TO 20 DO
	gvl.motorDrive[i].StatusDisplay();
	gvl.motorDrive[i].CalculateMotorAngle();
	gvl.motorDrive[i].CalibrateTrqData();
END_FOR

// Axis level 
// Group command handling,批量控制，需调用单轴控制实现
gvl.uiHandler.GroupMotionCmdHandling();
gvl.uiHandler.GroupForceCtrlCmdHandling();
// Axis command handling,单轴运动控制和力控
gvl.uiHandler.AxisMotionCmdHandling();
gvl.uiHandler.AxisForceCtrlCmdHandling();
// TrqSensor command handling,扭矩传感器清零
gvl.uiHandler.TrqSensorCmdHandling();
// gait command handling步态控制
gvl.uiHandler.GaitCtrlCmdHandling();

// receive imu data from ads
(*gvl.accx := gvl.IMUDATA[1];
gvl.accy := gvl.IMUDATA[2];
gvl.accz := gvl.IMUDATA[3];
gvl.roll := gvl.IMUDATA[4];
gvl.pitch := gvl.IMUDATA[5];
gvl.yaw  := gvl.IMUDATA[6];

// update robot states
gvl.rpy_model[0] := gvl.roll/180.0*pi;
gvl.rpy_model[1] := gvl.pitch/180.0*pi;
gvl.rpy_model[2] := gvl.yaw/180.0*pi;*)
gvl.roll := gvl.rpy_inpt[0];
gvl.pitch := gvl.rpy_inpt[1];
gvl.yaw  := gvl.rpy_inpt[2];
gvl.rpy_model[0] := gvl.roll/180.0*pi;
gvl.rpy_model[1] := gvl.pitch/180.0*pi;
gvl.rpy_model[2] := gvl.yaw/180.0*pi;


FOR i := 0 TO 5 DO
	FOR j := 0 TO 2 DO
		gvl.legCtrl[i].UpdateDriveFeedbacks(gvl.motorDrive[i*3 + j], j,i);////yk 调用18次，每次调用写入一次腿运动学参数
	END_FOR
	
	gvl.legCtrl[i].ForwardKinetics(
		motorAngles := gvl.legCtrl[i].motorAnglesIn,
		legIndex:=i,
		tipPosition => tipPos);
		
	gvl.legCtrl[i].TipVelocity(
		motorVel := gvl.legCtrl[i].motorAngVelIn,
		motorAng := gvl.legCtrl[i].motorAnglesIn,
		legIndex:=i,
		tipVel   => tipVel);
		
	gvl.legCtrl[i].TipForce(
		motorTrq := gvl.legCtrl[i].jointTorqueIn,
		motorAng := gvl.legCtrl[i].motorAnglesIn,
		legIndex:=i,
		tipFce   => tipFce);
		
	FOR j := 0 TO 2 DO
		gvl.tipActualPos[i, j] := tipPos[j];
		gvl.tipActualVel[i, j] := tipVel[j];
		gvl.tipActualFce[i, j] := tipFce[j];
		gvl.jntActualPos[i, j] := gvl.legCtrl[i].motorAnglesIn[j];
		gvl.jntActualVel[i, j] := gvl.legCtrl[i].motorAngVelIn[j];
		gvl.jntActualFce[i, j] := gvl.legCtrl[i].jointTorqueIn[j];
		gvl.jntLastRefPos[i, j] := gvl.legCtrl[i].motorRefAnglesIn[j];
	END_FOR
END_FOR

///////////////////////////////////////////////////////
// Gait Control

IF gvl.isInGaitMode THEN
	gvl.gaitPlanner.DoPlanning(isDone => gvl.isFinished); 
	
	IF gvl.isFinished OR gvl.emergencyStop THEN
		gvl.gaitPlanner.FinalizeGaitCmd();
		gvl.isInGaitMode := FALSE;
	END_IF
	
	// Download cmds
	FOR i := 0 TO 5 DO
		// copy cmds to each leg,
		gvl.legCtrl[i].SetReference();
		// map ref pos, vel, and fce to actual joints
		FOR j := 0 TO 2 DO
			gvl.legCtrl[i].DownloadDriveCmds(gvl.motorDrive[i*3 + j], j,i);
		END_FOR
	END_FOR
END_IF

// Drive level control
FOR i := 0 TO 20 DO	
	// Mid level control algorithms
	IF NOT gvl.motorDrive[i].isInForceControl THEN
		IF i=18 OR i=19 OR i=20 THEN
			gvl.opModeCmd[i] := 3;
		ELSE
			gvl.opModeCmd[i] := 9;
		END_IF
		IF i=20 THEN
			IF gvl.motorDrive[i].IsAbsMoveState=TRUE THEN
				gvl.opModeCmd[i] := 1;
			ELSE
				gvl.opModeCmd[i] := 3;				
			END_IF
		END_IF
		
		gvl.motorDrive[i].GoHome(); 
		gvl.motorDrive[i].JogControl();
		gvl.motorDrive[i].AbsMove();
	ELSE
		gvl.opModeCmd[i] := 10;
		gvl.motorDrive[i].ImpedControl(
			desiredTorque := 0,
			isExternalIC := FALSE);//阻抗参数已经通过gvl.legCtrl[i].DownloadDriveCmds(gvl.motorDrive[i*3 + j], j)写入，所以这里参考力为0
		
		//gvl.motorDrive[i].ImpedControl2();
		
		// Convert torque (Nm) to current cmd ( per 1/1000 )
		gvl.motorDrive[i].CalculateCurrentCmd();
	END_IF
	
	// Low level control
	gvl.motorDrive[i].DriverControl(gvl.opModeCmd[i], gvl.enableCmd[i]);
END_FOR


(*
yk 需要根据实际更新
// torque sensor board control
gvl.setCtrlZero[0] := 0;
gvl.setCtrlZero[1] := 0;
FOR i := 0 TO 11 DO
	IF i < 6 THEN
		gvl.setCtrlZero[0] := gvl.setCtrlZero[0] OR SHL(gvl.motorDrive[i].trqSensor.reqReset, 5 - i);
	ELSE
		gvl.setCtrlZero[1] := gvl.setCtrlZero[1] OR SHL(gvl.motorDrive[i].trqSensor.reqReset, i - 6);
	END_IF
END_FOR
*)

// clear emergency stop event
IF gvl.emergencyStop THEN
	// count emergency stop event number
	gvl.emergencyStopCount := gvl.emergencyStopCount+1;
	// clear
	gvl.emergencyStop := FALSE;
END_IF

FOR i:=0 TO 5 DO
	FOR j:=0 TO 2 DO
		gvl.jntRefVelDif[i,j]:=(gvl.jntRefPos[i,j]-gvl.lastjntRefPos[i,j])*DINT_TO_LREAL(gvl.sampleRate);
		gvl.lastjntRefPos[i,j]:=gvl.jntRefPos[i,j];
	END_FOR
END_FOR

IF gvl.setRcRefAngButton=TRUE THEN
	gvl.jntRefPosLastPlanning:=gvl.jntRefPosLastPlanningFirstRc;
	gvl.setRcRefAngButton:=FALSE;
END_IF

IF gvl.RestButton=TRUE AND gvl.WorkButton=FALSE THEN
	gvl.ReduceDistance:=-0.08;
	gvl.IsRest:=TRUE;
	gvl.IsWork:=FALSE;
	gvl.LiftBodyStartFlag:=TRUE;
	gvl.LiftBodyEndFlag:=FALSE;
	gvl.LiftBodyEndFlagLast:=FALSE;
	gvl.RestButton:=FALSE;
END_IF
IF gvl.RestButton=FALSE AND gvl.WorkButton=TRUE THEN
	gvl.ReduceDistance:=0.08;
	gvl.IsWork:=TRUE;
	gvl.IsRest:=FALSE;
	gvl.LiftBodyStartFlag:=TRUE;
	gvl.LiftBodyEndFlag:=FALSE;
	gvl.LiftBodyEndFlagLast:=FALSE;
	gvl.WorkButton:=FALSE;
END_IF

IF gvl.IsRest=TRUE THEN
	IF gvl.LiftBodyStartFlag=TRUE THEN
		gvl.LiftBodyStartFlag:=FALSE;
		gvl.gaitId:=2;
		gvl.IsLiftBody:=TRUE;
		IF gvl.ReduceDistance>0 THEN
			gvl.ReduceDistance:=-gvl.ReduceDistance;
		END_IF
		IF ABS(gvl.ReduceDistance)>=0.15 THEN
			gvl.ReduceDistance:=-0.15;
		END_IF 
		GVL.startGaitButton:=TRUE;
		gvl.LiftBodyStartFlag:=FALSE;
		gvl.LiftBodyEndFlag:=FALSE;
	END_IF
	IF gvl.IsLiftBody:=TRUE AND GVL.isInGaitMode=TRUE THEN
		gvl.LiftBodyEndFlag:= gvl.isFinished;
	END_IF	
	IF gvl.LiftBodyEndFlagLast=FALSE AND gvl.LiftBodyEndFlag=TRUE AND gvl.IsLiftBody=TRUE THEN
		gvl.IsLiftBody:=FALSE;
		gvl.IsRest:=FALSE;
	END_IF
	gvl.LiftBodyEndFlagLast:=gvl.LiftBodyEndFlag;	
END_IF

IF gvl.IsWork=TRUE THEN
	IF gvl.LiftBodyStartFlag=TRUE THEN
		gvl.LiftBodyStartFlag:=FALSE;
		gvl.gaitId:=2;
		gvl.IsLiftBody:=TRUE;
		IF gvl.ReduceDistance<0 THEN
			gvl.ReduceDistance:=-gvl.ReduceDistance;
		END_IF
		IF ABS(gvl.ReduceDistance)>=0.15 THEN
			gvl.ReduceDistance:=0.15;
		END_IF 
		GVL.startGaitButton:=TRUE;
		gvl.LiftBodyStartFlag:=FALSE;
		gvl.LiftBodyEndFlag:=FALSE;
	END_IF
	IF gvl.IsLiftBody:=TRUE AND GVL.isInGaitMode=TRUE THEN
		gvl.LiftBodyEndFlag:= gvl.isFinished;
	END_IF	
	IF gvl.LiftBodyEndFlagLast=FALSE AND gvl.LiftBodyEndFlag=TRUE AND gvl.IsLiftBody=TRUE THEN
		gvl.IsLiftBody:=FALSE;
		gvl.IsWork:=FALSE;
	END_IF
	gvl.LiftBodyEndFlagLast:=gvl.LiftBodyEndFlag;	
END_IF

END_PROGRAM

// ---- POUs/UIHandler.TcPOU
FUNCTION_BLOCK UIHandler
VAR_INPUT
END_VAR
VAR_OUTPUT
END_VAR
VAR
	zeroSetCount : DINT := 500;
END_VAR

METHOD PUBLIC AxisForceCtrlCmdHandling : BOOL
VAR_INPUT
END_VAR

VAR
	i: INT;
END_VAR
// Axis command handling
FOR i := 0 TO 17 DO	
	(*IF gvl.emergencyStop THEN
		gvl.axisForceCtrlButton[i] := FALSE;
	END_IF*)
	
	IF GVL.axisForceCtrlButton[i] THEN
		IF NOT gvl.axisForceCtrlModeInd[i] THEN
			gvl.motorDrive[i].startForceControl();
			IF gvl.motorDrive[i].isInForceControl THEN
				gvl.axisForceCtrlModeInd[i] := TRUE;
			ELSE
				gvl.axisForceCtrlButton[i] := FALSE;
			END_IF
		END_IF
	ELSE
		IF gvl.axisForceCtrlModeInd[i] THEN
			gvl.axisForceCtrlModeInd[i] := FALSE;
			gvl.motorDrive[i].StopForceControl();
		END_IF
	END_IF
	
END_FOR
END_METHOD

METHOD PUBLIC AxisMotionCmdHandling : BOOL
VAR_INPUT
END_VAR

VAR
	i: INT;
END_VAR
// Axis command handling,轴的运动最后都通过主函数调用JogControll函数实现，设置home位置，通过主函数调用电机驱动函数实现
FOR i := 0 TO 20 DO	

	IF GVL.enableButton[i] THEN
		GVL.enablebuttonText[i] :='Power Off';
	ELSE
		GVL.enablebuttonText[i] :='Power On';
	END_IF
	
	IF gvl.setInitPositionButton[i] THEN
		gvl.motorDrive[i].SetInitPosition();
		gvl.setInitPositionButton[i] := FALSE;
	END_IF
	
	IF gvl.startHomeButton[i] THEN
		gvl.motorDrive[i].StartGoHome();
		gvl.startHomeButton[i] := FALSE;
	END_IF
	
	IF gvl.AbsMoveButton[i] THEN
		gvl.motorDrive[i].StartAbsMove(GVL.AbsMoveTgtPos[i]);
		gvl.AbsMoveButton[i] := FALSE;
	END_IF
	
	IF gvl.AbsMoveStopButton[i] THEN
		gvl.motorDrive[i].StopAbsMove();
		gvl.AbsMoveStopButton[i] := FALSE;
	END_IF
	
	IF gvl.jogButton[i] THEN
		gvl.motorDrive[i].StartJog(gvl.jogVelocity[i]);
		gvl.jogButton[i] := FALSE;
	END_IF
	
	IF gvl.jogStopButton[i] THEN
		gvl.motorDrive[i].StopJog();
		gvl.jogStopButton[i] := FALSE;
	END_IF
	
	gvl.enableCmd[i] := GVL.enableButton[i]; 
END_FOR
END_METHOD

METHOD PUBLIC GaitCtrlCmdHandling : BOOL
VAR_INPUT
END_VAR
IF gvl.startGaitButton AND NOT gvl.isInGaitMode THEN
	gvl.gaitPlanner.Initialize();
	gvl.isInGaitMode := TRUE;
	gvl.startGaitButton := FALSE;
	gvl.isFinished := FALSE;
END_IF
END_METHOD

METHOD PUBLIC GroupForceCtrlCmdHandling : BOOL
VAR_INPUT
END_VAR

VAR
	i: INT;
END_VAR
IF gvl.forceCtrlGroupButton THEN
	FOR i:= 0 TO 17 DO
		IF gvl.activeAxisList[gvl.groupSelector][i] = 1 THEN
			gvl.axisForceCtrlButton[i] := TRUE;
		END_IF
	END_FOR
	gvl.forceCtrlGroupButton := FALSE;
END_IF

IF gvl.forceCtrlGroupOffButton THEN
	FOR i:= 0 TO 17 DO
		IF gvl.activeAxisList[gvl.groupSelector][i] = 1 THEN
			gvl.axisForceCtrlButton[i] := FALSE;
		END_IF
	END_FOR
	gvl.forceCtrlGroupOffButton := FALSE;
END_IF

IF gvl.useHardImpedButton THEN
	gvl.kpGroup := 2000;
	gvl.kdGroup := 200;
	gvl.kpTrqGroup := 0;
	gvl.kiTrqGroup := 0;
	gvl.useParamIndex := 1;
	gvl.useHardImpedButton := FALSE;
END_IF

IF gvl.useSoftImpedButton THEN
	gvl.kpGroup := 220;
	gvl.kdGroup := 25;
	gvl.kpTrqGroup := 0.65;
	gvl.kiTrqGroup := 0.5;
	gvl.useParamIndex := 0;
	gvl.useSoftImpedButton := FALSE;
END_IF

IF gvl.setGroupImpedButton THEN
	FOR i:= 0 TO 17 DO
		gvl.motorDrive[i].SetImpedanceParam(gvl.kpGroup, gvl.kdGroup, gvl.kpTrqGroup, gvl.kiTrqGroup);
	END_FOR
	gvl.setGroupImpedButton := FALSE;
END_IF
END_METHOD

METHOD PUBLIC GroupMotionCmdHandling : BOOL
VAR_INPUT
END_VAR
VAR_OUTPUT
END_VAR
VAR
	i: INT;
END_VAR
IF gvl.enableGroupButton THEN
	FOR i:= 0 TO 17 DO
		IF gvl.activeAxisList[gvl.groupSelector][i] = 1 THEN
			gvl.enableButton[i] := TRUE;
		END_IF
	END_FOR
	gvl.enableButton[18] := TRUE;
	gvl.enableButton[19] := TRUE;
	gvl.enableButton[20] := TRUE;
	gvl.enableGroupButton := FALSE;
END_IF

IF gvl.disableGroupButton THEN
	FOR i:= 0 TO 17 DO
		IF gvl.activeAxisList[gvl.groupSelector][i] = 1 THEN
			gvl.enableButton[i] := FALSE;
		END_IF
	END_FOR
	gvl.enableButton[18] := FALSE;
	gvl.enableButton[19] := FALSE;
	gvl.enableButton[20] := FALSE;
	gvl.disableGroupButton := FALSE;
END_IF

IF gvl.homeGroupButton THEN
	FOR i:= 0 TO 17 DO
		IF gvl.activeAxisList[gvl.groupSelector][i] = 1 THEN
			gvl.startHomeButton[i] := TRUE;
		END_IF
	END_FOR
	gvl.homeGroupButton := FALSE;
END_IF

IF gvl.setPosGroupButton THEN
	FOR i:= 0 TO 17 DO
		IF gvl.activeAxisList[gvl.groupSelector][i] = 1 THEN
			gvl.setInitPositionButton[i] := TRUE;
		END_IF
	END_FOR
	gvl.setPosGroupButton := FALSE;
END_IF

IF gvl.jogGroupButton THEN
	FOR i:= 0 TO 17 DO
		IF gvl.activeAxisList[gvl.groupSelector][i] = 1 THEN
			gvl.jogButton[i] := TRUE;
			gvl.jogVelocity[i] := gvl.jogGroupVelocity;
		END_IF
	END_FOR
	gvl.jogGroupButton := FALSE;
END_IF

IF gvl.jogStopGroupButton THEN
	FOR i:= 0 TO 17 DO
		IF gvl.activeAxisList[gvl.groupSelector][i] = 1 THEN
			gvl.jogStopButton[i] := TRUE;
		END_IF
	END_FOR
	gvl.jogStopGroupButton := FALSE;
END_IF
END_METHOD

METHOD PUBLIC Initialize : BOOL
VAR_INPUT
END_VAR

VAR
	i: INT;
END_VAR
FOR i := 0 TO 19 DO
	gvl.enableButton[i] := FALSE;
	gvl.startHomeButton[i] := FALSE;
	gvl.setInitPositionButton[i] := FALSE; //yk 设置home位置,home结束需要点击setposition写入
	gvl.jogButton[i] := FALSE;
	gvl.jogVelocity[i] := 0.05;
	gvl.axisForceCtrlButton[i] := FALSE;  //yk 切换为力控模式
	gvl.axisForceCtrlModeInd[i] := FALSE;//yk 指示灯是否力控
END_FOR
END_METHOD

METHOD PUBLIC TrqSensorCmdHandling : BOOL
VAR_INPUT
END_VAR
// TSR control
IF gvl.setTSRZeroButton THEN
	gvl.setTrqSensorZero[0] := 63;
	gvl.setTrqSensorZero[1] := 63;
	gvl.setTrqSensorZero[2] := 63;
	zeroSetCount := zeroSetCount - 1;
ELSE
	gvl.setTrqSensorZero[0] := 0;
	gvl.setTrqSensorZero[1] := 0;
	gvl.setTrqSensorZero[2] := 0;
	zeroSetCount := 500;
END_IF

//往力传感器发送500次清零，防止丢包
IF zeroSetCount <= 0 THEN
	gvl.setTSRZeroButton := FALSE;
END_IF
END_METHOD

END_FUNCTION_BLOCK

// ---- POUs/GaitPlanner/GaitPlanner.TcPOU
FUNCTION_BLOCK GaitPlanner
VAR_INPUT
END_VAR
VAR_OUTPUT
END_VAR
VAR
	gaitCount : UDINT := 0;
	recoverGaitPlanner : RecoverGait;
	StaticwalkGaitPlanner    : StaticWalkGait;
	liftBodyGaitPlanner    : LiftBodyGait;
	swingBodyGaitPlanner : SwingBodyGait;
	CurlingGaitPlanner :CurlingGait;
	CurlingGaitPlanner2 :CurlingGaitFromStance;
	RcToSlipFromCurlingPlanner:RcToSlipFromCurling;
	BLegSlipPlanner:BLegSlip;
	CurlingGaitFromSlipPlanner:CurlingGaitFromSlip;
	RcToCurlingFromSlipPlanner:RcToCurlingFromSlip;
	RcToStanceFromSlipPlanner:RcToStanceFromSlip;
	TrotWalkPlanner:TrotWalk;
	WalkSlopePlanner : WalkSlopeGait;
	
	
END_VAR

METHOD PUBLIC DoPlanning : BOOL
VAR_INPUT
END_VAR
VAR_OUTPUT
	isDone : BOOL;
END_VAR

VAR
	i: INT;
	j: INT;
END_VAR
IF gvl.gaitId = 0 THEN
	recoverGaitPlanner.DoPlanning(gaitCount);
	isDone := recoverGaitPlanner.isFinished;
	FOR i := 0 TO 5 DO
		FOR j := 0 TO 2 DO
			gvl.jntRefPosTuning[i, j] := recoverGaitPlanner.jointPosTarget[i, j];
			gvl.jntRefVelTuning[i, j] := recoverGaitPlanner.jointVelTarget[i, j];
			gvl.jntRefFceTuning[i, j] := recoverGaitPlanner.jointFceTarget[i, j];
		END_FOR
	END_FOR
ELSIF gvl.gaitId = 1 THEN
	StaticwalkGaitPlanner.DoPlanning(gaitCount);
	isDone := StaticwalkGaitPlanner.isFinished;
	FOR i := 0 TO 5 DO
		FOR j := 0 TO 2 DO
			gvl.jntRefPosTuning[i, j] := StaticwalkGaitPlanner.jointPosTarget[i, j];
			gvl.jntRefVelTuning[i, j] := StaticwalkGaitPlanner.jointVelTarget[i, j];
			gvl.jntRefFceTuning[i, j] := StaticwalkGaitPlanner.jointFceTarget[i, j];
		END_FOR
	END_FOR
ELSIF gvl.gaitId = 2 THEN
	liftBodyGaitPlanner.DoPlanning(count:=gaitCount );
	isDone := liftBodyGaitPlanner.isFinished;
	FOR i := 0 TO 5 DO
		FOR j := 0 TO 2 DO
			gvl.jntRefPosTuning[i, j] := liftBodyGaitPlanner.jointPosTarget[i, j];
			gvl.jntRefVelTuning[i, j] := liftBodyGaitPlanner.jointVelTarget[i, j];
			gvl.jntRefFceTuning[i, j] := liftBodyGaitPlanner.jointFceTarget[i, j];
		END_FOR
	END_FOR	

ELSIF gvl.gaitId = 3 THEN
	swingBodyGaitPlanner.DoPlanning(gaitCount);
	isDone := swingBodyGaitPlanner.isFinished;
	FOR i := 0 TO 5 DO
		FOR j := 0 TO 2 DO
			gvl.jntRefPosTuning[i, j] := swingBodyGaitPlanner.jointPosTarget[i, j];
			gvl.jntRefVelTuning[i, j] := swingBodyGaitPlanner.jointVelTarget[i, j];
			gvl.jntRefFceTuning[i, j] := swingBodyGaitPlanner.jointFceTarget[i, j];
		END_FOR
	END_FOR
ELSIF gvl.gaitId = 4 THEN
	CurlingGaitPlanner2.DoPlanning(gaitCount);
	isDone := CurlingGaitPlanner2.isFinished;
	FOR i := 0 TO 5 DO
		FOR j := 0 TO 2 DO
			gvl.jntRefPosTuning[i, j] := CurlingGaitPlanner2.jointPosTarget[i, j];
			gvl.jntRefVelTuning[i, j] := CurlingGaitPlanner2.jointVelTarget[i, j];
			gvl.jntRefFceTuning[i, j] := CurlingGaitPlanner2.jointFceTarget[i, j];
		END_FOR
	END_FOR
ELSIF gvl.gaitId = 5 THEN
	CurlingGaitFromSlipPlanner.DoPlanning(gaitCount);
	isDone := CurlingGaitFromSlipPlanner.isFinished;
	FOR i := 0 TO 5 DO
		FOR j := 0 TO 2 DO
			gvl.jntRefPosTuning[i, j] := CurlingGaitFromSlipPlanner.jointPosTarget[i, j];
			gvl.jntRefVelTuning[i, j] := CurlingGaitFromSlipPlanner.jointVelTarget[i, j];
			gvl.jntRefFceTuning[i, j] := CurlingGaitFromSlipPlanner.jointFceTarget[i, j];
		END_FOR
	END_FOR
ELSIF gvl.gaitId = 6 THEN
	RcToSlipFromCurlingPlanner.DoPlanning(gaitCount);
	isDone := RcToSlipFromCurlingPlanner.isFinished;
	FOR i := 0 TO 5 DO
		FOR j := 0 TO 2 DO
			gvl.jntRefPosTuning[i, j] := RcToSlipFromCurlingPlanner.jointPosTarget[i, j];
			gvl.jntRefVelTuning[i, j] := RcToSlipFromCurlingPlanner.jointVelTarget[i, j];
			gvl.jntRefFceTuning[i, j] := RcToSlipFromCurlingPlanner.jointFceTarget[i, j];
		END_FOR
	END_FOR
ELSIF gvl.gaitId = 7 THEN
	RcToCurlingFromSlipPlanner.DoPlanning(gaitCount);
	isDone := RcToCurlingFromSlipPlanner.isFinished;
	FOR i := 0 TO 5 DO
		FOR j := 0 TO 2 DO
			gvl.jntRefPosTuning[i, j] := RcToCurlingFromSlipPlanner.jointPosTarget[i, j];
			gvl.jntRefVelTuning[i, j] := RcToCurlingFromSlipPlanner.jointVelTarget[i, j];
			gvl.jntRefFceTuning[i, j] := RcToCurlingFromSlipPlanner.jointFceTarget[i, j];
		END_FOR
	END_FOR
ELSIF gvl.gaitId = 8 THEN
	RcToStanceFromSlipPlanner.DoPlanning(gaitCount);
	isDone := RcToStanceFromSlipPlanner.isFinished;
	FOR i := 0 TO 5 DO
		FOR j := 0 TO 2 DO
			gvl.jntRefPosTuning[i, j] := RcToStanceFromSlipPlanner.jointPosTarget[i, j];
			gvl.jntRefVelTuning[i, j] := RcToStanceFromSlipPlanner.jointVelTarget[i, j];
			gvl.jntRefFceTuning[i, j] := RcToStanceFromSlipPlanner.jointFceTarget[i, j];
		END_FOR
	END_FOR
ELSIF gvl.gaitId = 9 THEN
	BLegSlipPlanner.DoPlanning(gaitCount);
	isDone := BLegSlipPlanner.isFinished;
	FOR i := 0 TO 5 DO
		FOR j := 0 TO 2 DO
			gvl.jntRefPosTuning[i, j] := BLegSlipPlanner.jointPosTarget[i, j];
			gvl.jntRefVelTuning[i, j] := BLegSlipPlanner.jointVelTarget[i, j];
			gvl.jntRefFceTuning[i, j] := BLegSlipPlanner.jointFceTarget[i, j];
		END_FOR
	END_FOR
ELSIF gvl.gaitId = 10 THEN
	TrotWalkPlanner.DoPlanning(gaitCount);
	isDone := TrotWalkPlanner.isFinished;
	FOR i := 0 TO 5 DO
		FOR j := 0 TO 2 DO
			gvl.jntRefPosTuning[i, j] := TrotWalkPlanner.jointPosTarget[i, j];
			gvl.jntRefVelTuning[i, j] := TrotWalkPlanner.jointVelTarget[i, j];
			gvl.jntRefFceTuning[i, j] := TrotWalkPlanner.jointFceTarget[i, j];
		END_FOR
	END_FOR
ELSIF gvl.gaitId = 11 THEN
	WalkSlopePlanner.DoPlanning(gaitCount);
	isDone := WalkSlopePlanner.isFinished;
	FOR i := 0 TO 5 DO
		FOR j := 0 TO 2 DO
			gvl.jntRefPosTuning[i, j] := WalkSlopePlanner.jointPosTarget[i, j];
			gvl.jntRefVelTuning[i, j] := WalkSlopePlanner.jointVelTarget[i, j];
			gvl.jntRefFceTuning[i, j] := WalkSlopePlanner.jointFceTarget[i, j];
		END_FOR
	END_FOR
ELSE
	// no gait selected
	FOR i := 0 TO 5 DO
		FOR j := 0 TO 2 DO
			IF ABS(gvl.jntActualPos[i, j]-gvl.lastjntRefPos[i,j])<0.1 THEN
				gvl.jntRefPosTuning[i, j] :=gvl.lastjntRefPos[i,j];
			ELSE
				gvl.jntRefPosTuning[i, j] := gvl.jntActualPos[i, j];				
			END_IF
			gvl.jntRefVelTuning[i, j] := 0;
			gvl.jntRefFceTuning[i, j] := 0;
		END_FOR
	END_FOR
	isDone := TRUE;
END_IF

//Tuning state 
(*FOR i := 0 TO 5 DO
	FOR j := 0 TO 2 DO
			IF ABS(gvl.jntActualPos[i, j]-gvl.lastjntRefPos[i,j])<0.1 THEN
				gvl.jntRefPos[i, j] :=gvl.lastjntRefPos[i,j];
			ELSE
				gvl.jntRefPos[i, j] := gvl.jntActualPos[i, j];				
			END_IF
		gvl.jntRefVel[i, j] := 0;
		gvl.jntRefFce[i, j] := 0;
	END_FOR
END_FOR*)

//Actual employment
gvl.jntRefPos:=gvl.jntRefPosTuning;
gvl.jntRefVel:=gvl.jntRefVelTuning;
gvl.jntRefFce:=gvl.jntRefFceTuning;

gaitCount := gaitCount + 1;
END_METHOD

METHOD PUBLIC FinalizeGaitCmd : BOOL
VAR_INPUT
END_VAR

VAR
	i: INT;
	j: INT;
END_VAR
FOR i := 0 TO 5 DO
	FOR j := 0 TO 2 DO
		//gvl.jntRefPos[i, j] := gvl.jntActualPos[i, j];
		gvl.jntRefVel[i, j] := 0;
		gvl.jntRefFce[i, j] := 0;
	END_FOR
END_FOR
END_METHOD

METHOD PUBLIC Initialize : BOOL
VAR_INPUT
END_VAR
gaitCount := 0;
END_METHOD

END_FUNCTION_BLOCK

// ---- POUs/GaitPlanner/RecoverGait.TcPOU
FUNCTION_BLOCK RecoverGait
VAR_INPUT
END_VAR
VAR_OUTPUT
END_VAR
VAR
	isFinished : BOOL := FALSE;
	tRetract   : LREAL := 3;
	tWait      : LREAL := 1;
	tExtend    : LREAL := 3;
	jntAngStart:ARRAY[0..5,0..2] OF LREAL;
	jntAngRetract0:ARRAY[0..5,0..2] OF LREAL:=[0,150.7997*pi/180,291.8958*pi/180,
											  0,327.8142*pi/180,(196.8366-327.8142)*pi/180,
											  0,172.5134*pi/180,(269.4767-172.5134)*pi/180,
											  0,172.5134*pi/180,(269.4767-172.5134)*pi/180,
											  0,327.8142*pi/180,(196.8366-327.8142)*pi/180,
											  0,150.7997*pi/180,291.8958*pi/180];//walk
	jntAngRetract1:ARRAY[0..5,0..2] OF LREAL:=[0,163.1808*pi/180,297.208*pi/180,
											  0,322.9120*pi/180,(205.1705-322.9120)*pi/180,
											  0,183.8227*pi/180,(269.8634-183.8227)*pi/180,
											  0,183.8227*pi/180,(269.8634-183.8227)*pi/180,
											  0,322.9120*pi/180,(205.1705-322.9120)*pi/180,
											  0,163.1808*pi/180,297.208*pi/180];//curling	
	jntAngRetract:ARRAY[0..5,0..2] OF LREAL	;								  

	jntAngExtend0:ARRAY[0..5,0..2] OF LREAL:=[0,163.1808*pi/180,297.208*pi/180,
											 0,320.9331*pi/180,(208.0880-320.9331)*pi/180,	
											 0,187.8384*pi/180,(269.4264-187.8384)*pi/180,
											 0,187.8384*pi/180,(269.4264-187.8384)*pi/180,
									         0,320.9331*pi/180,(208.0880-320.9331)*pi/180,
											 0,163.1808*pi/180,297.208*pi/180];//walk
	jntAngExtend1:ARRAY[0..5,0..2] OF LREAL:=[0,181.9845*pi/180,299.9603*pi/180,
											 0,302.7132*pi/180,(230.9946-302.7132)*pi/180,	
											 0,222.0252*pi/180,(254.0072-222.0252)*pi/180,
											 0,222.0252*pi/180,(254.0072-222.0252)*pi/180,
									         0,302.7132*pi/180,(230.9946-302.7132)*pi/180,
											 0,181.9845*pi/180,299.9603*pi/180];//curling
	jntAngExtend:ARRAY[0..5,0..2] OF LREAL;										 
											 
										 
	pivot, pivotDot : LREAL;
	getPivot  : GetPivot;	
	fbGetPivot  : GetPivot;
	pvt, pvtDot : LREAL;

	jointPosTarget  : ARRAY[0..5, 0..2] OF LREAL; 
	jointVelTarget  : ARRAY[0..5, 0..2] OF LREAL;  
	jointFceTarget  : ARRAY[0..5, 0..2] OF LREAL;	

	tipForceDesire:ARRAY[0..5,0..2] OF LREAL;
	jntTrqDesire:ARRAY[0..5,0..2] OF LREAL;
	fceLoadTime:LREAL:=0.5;
	tipForceDesireGroupA:ARRAY[0..5,0..2] OF LREAL:=[0,-125,0,
													 0,0,0,
													 0,0,0,
													 0,0,0,
													 0,0,0,
													 0,0,0];
	tipForceDesireGroupB:ARRAY[0..5,0..2] OF LREAL:=[0,0,0,
													 0,0,0,
													 0,0,0,
													 0,0,0,
													 0,0,0,
													 0,-145,0];
	tipForceDesireZeros:ARRAY[0..5,0..2] OF LREAL:=[0,0,0,
													 0,0,0,
													 0,0,0,
													 0,0,0,
													 0,0,0,
													 0,0,0];								 
											 
END_VAR

METHOD PUBLIC DoPlanning : BOOL
VAR_INPUT
		count : UDINT;
END_VAR
VAR
	tTotal: LREAL;
	tNow: LREAL;
	tr:LREAL;
	
	jntPosBegin : ARRAY[0..5, 0..2] OF LREAL;
	jntPosEnd   : ARRAY[0..5, 0..2] OF LREAL;
	
	legExtractRefPosCurling: ARRAY[0..5, 0..2] OF LREAL:=[-0.35,-0.3+0.02,0,
														  0.1,-0.3+0.02,-0.1246,
														  -0.3+0.05,-0.3+0.02,-0.1246,
														  -0.3+0.05,-0.3+0.02,0.1246,
														  0.1,-0.3+0.02,0.1246,
														  -0.35,-0.3+0.02,0];//-0.15 for front leg
	jntExtractRefPosCurling: ARRAY[0..5, 0..2] OF LREAL:=[0,163.1808*pi/180,297.208*pi/180,
											  			  0,322.9120*pi/180,(205.1705-322.9120)*pi/180,
											              0,183.8227*pi/180,(269.8634-183.8227)*pi/180,
											              0,183.8227*pi/180,(269.8634-183.8227)*pi/180,
											              0,322.9120*pi/180,(205.1705-322.9120)*pi/180,
											              0,163.1808*pi/180,297.208*pi/180];
														  
	(*legExtendRefPosCurling: ARRAY[0..5, 0..2] OF LREAL:=[-0.35,-0.3805-0.07,0,
														  0.1,-0.4-0.07,-0.1246,
														  -0.3,-0.4-0.07,-0.1246,
														  -0.3,-0.4-0.07,0.1246,
														  0.1,-0.4-0.07,0.1246,
														  -0.35,-0.3805-0.07,0];//before change tip*)
	legExtendRefPosCurling: ARRAY[0..5, 0..2] OF LREAL:=[-0.35,-0.4-0.07,0,
														  0.1,-0.4-0.07,-0.1246,
														  -0.3+0.05,-0.4-0.07,-0.1246,
														  -0.3+0.05,-0.4-0.07,0.1246,
														  0.1,-0.4-0.07,0.1246,
														  -0.35,-0.4-0.07,0];//-0.15 for front leg														 
	
	jntExtendRefPosCurling: ARRAY[0..5, 0..2] OF LREAL:=[0,181.9845*pi/180,299.9603*pi/180,
											 			 0,302.7132*pi/180,(230.9946-302.7132)*pi/180,	
											             0,222.0252*pi/180,(254.0072-222.0252)*pi/180,
											             0,222.0252*pi/180,(254.0072-222.0252)*pi/180,
									                     0,302.7132*pi/180,(230.9946-302.7132)*pi/180,
											             0,181.9845*pi/180,299.9603*pi/180]	;	
									  
	legExtractRefPosWalk:    ARRAY[0..5, 0..2] OF LREAL:=[-0.35,-0.3+0.08,0,
														  0.1,-0.3209+0.08,-0.1246,
														  -0.3+0.05,-0.3209+0.08,-0.1246,
														  -0.3+0.05,-0.3209+0.08,0.1246,
														  0.1,-0.3209+0.08,0.1246,
														  -0.35,-0.3+0.08,0];	
														  
	jntExtractRefPosWalk: ARRAY[0..5, 0..2] OF LREAL:= [0,150.7997*pi/180,291.8958*pi/180,
											  			0,327.8142*pi/180,(196.8366-327.8142)*pi/180,
											  			0,172.5134*pi/180,(269.4767-172.5134)*pi/180,
											  			0,172.5134*pi/180,(269.4767-172.5134)*pi/180,
											  			0,327.8142*pi/180,(196.8366-327.8142)*pi/180,
											  			0,150.7997*pi/180,291.8958*pi/180];													  
														  
	(*legExtendRefPosWalk: ARRAY[0..5, 0..2] OF LREAL    :=[-0.35,-0.3,0,
														  0.1,-0.3209,-0.1246,
														  -0.3,-0.3209,-0.1246,
														  -0.3,-0.3209,0.1246,
														  0.1,-0.3209,0.1246,
														  -0.35,-0.3,0];//before change tip*)
	legExtendRefPosWalk: ARRAY[0..5, 0..2] OF LREAL    :=[-0.35,-0.3209,0,
														  0.1,-0.3209,-0.1246,
														  -0.3+0.05,-0.3209,-0.1246,
														  -0.3+0.05,-0.3209,0.1246,
														  0.1,-0.3209,0.1246,
														  -0.35,-0.3209,0];														  
														  
														  
	jntExtendRefPosWalk: ARRAY[0..5, 0..2] OF LREAL:=	   [0,163.1808*pi/180,297.208*pi/180,
											 				0,320.9331*pi/180,(208.0880-320.9331)*pi/180,	
											 				0,187.8384*pi/180,(269.4264-187.8384)*pi/180,
															0,187.8384*pi/180,(269.4264-187.8384)*pi/180,
									         				0,320.9331*pi/180,(208.0880-320.9331)*pi/180,
											 				0,163.1808*pi/180,297.208*pi/180];																						 
	i: INT;
	j: INT;
	tempLeg:ARRAY [0..2] OF LREAL;
	tempJnt:ARRAY [0..2] OF LREAL;
	tempRef:ARRAY [0..2] OF LREAL;
	
	tempTipForce:ARRAY [0..2] OF LREAL;
	temJntActPos:ARRAY [0..2] OF LREAL;
	tempDesJntTrq:ARRAY [0..2] OF LREAL;
END_VAR
IF count = 0 THEN
	isFinished := FALSE;
	FOR i:=0 TO 5 DO
		tempLeg[0]:=legExtractRefPosCurling[i,0];tempLeg[1]:=legExtractRefPosCurling[i,1];tempLeg[2]:=legExtractRefPosCurling[i,2];
		tempRef[0]:=jntExtractRefPosCurling[i,0];tempRef[1]:=jntExtractRefPosCurling[i,1];tempRef[2]:=jntExtractRefPosCurling[i,2];
		GVL.legCtrl[i].InverseKinetics(tipPosition:=tempLeg , refPosLast:=tempRef , legIndex:=i , motorAngles=>tempJnt , isSingular=> );
		jntAngRetract1[i,0]:=tempJnt[0];jntAngRetract1[i,1]:=tempJnt[1];jntAngRetract1[i,2]:=tempJnt[2];
		
		tempLeg[0]:=legExtractRefPosWalk[i,0];tempLeg[1]:=legExtractRefPosWalk[i,1];tempLeg[2]:=legExtractRefPosWalk[i,2];
		tempRef[0]:=jntExtractRefPosWalk[i,0];tempRef[1]:=jntExtractRefPosWalk[i,1];tempRef[2]:=jntExtractRefPosWalk[i,2];
		GVL.legCtrl[i].InverseKinetics(tipPosition:=tempLeg , refPosLast:=tempRef , legIndex:=i , motorAngles=>tempJnt , isSingular=> );
		jntAngRetract0[i,0]:=tempJnt[0];jntAngRetract0[i,1]:=tempJnt[1];jntAngRetract0[i,2]:=tempJnt[2];
		
		tempLeg[0]:=legExtendRefPosCurling[i,0];tempLeg[1]:=legExtendRefPosCurling[i,1];tempLeg[2]:=legExtendRefPosCurling[i,2];
		tempRef[0]:=jntExtendRefPosCurling[i,0];tempRef[1]:=jntExtendRefPosCurling[i,1];tempRef[2]:=jntExtendRefPosCurling[i,2];
		GVL.legCtrl[i].InverseKinetics(tipPosition:=tempLeg , refPosLast:=tempRef , legIndex:=i , motorAngles=>tempJnt , isSingular=> );
		jntAngExtend1[i,0]:=tempJnt[0];jntAngExtend1[i,1]:=tempJnt[1];jntAngExtend1[i,2]:=tempJnt[2];		
		
		tempLeg[0]:=legExtendRefPosWalk[i,0];tempLeg[1]:=legExtendRefPosWalk[i,1];tempLeg[2]:=legExtendRefPosWalk[i,2];
		tempRef[0]:=jntExtendRefPosWalk[i,0];tempRef[1]:=jntExtendRefPosWalk[i,1];tempRef[2]:=jntExtendRefPosWalk[i,2];
		GVL.legCtrl[i].InverseKinetics(tipPosition:=tempLeg , refPosLast:=tempRef , legIndex:=i , motorAngles=>tempJnt , isSingular=> );
		jntAngExtend0[i,0]:=tempJnt[0];jntAngExtend0[i,1]:=tempJnt[1];jntAngExtend0[i,2]:=tempJnt[2];		
	END_FOR
	
	IF gvl.RcGaitId=0 THEN
		jntAngRetract:=jntAngRetract0;
		jntAngExtend:=jntAngExtend0;
	ELSE
		jntAngRetract:=jntAngRetract1;
		jntAngExtend:=jntAngExtend1;			
	END_IF
	
	FOR i := 0 TO 5 DO
		FOR j := 0 TO 2 DO
			IF ABS(gvl.jntLastRefPos[i, j] - gvl.jntActualPos[i, j]) < 0.2 THEN
				jntAngStart[i,j] := gvl.jntLastRefPos[i, j];
			ELSE
				jntAngStart[i,j] := gvl.jntActualPos[i, j];
			END_IF
			jntAngStart[i,j]:=MinDistanceValue(jntAngStart[i,j],gvl.jntRefPosLastPlanning[i,j]);
			
		END_FOR
	END_FOR	
	
	tipForceDesire:=tipForceDesireZeros;	
END_IF

IF count<=(tRetract + tWait + tExtend) * gvl.sampleRate THEN //leg 0-2-4 recovery
	
//******************************force compensator******************************
	IF count<=fceLoadTime*gvl.sampleRate THEN
		tr  := UDINT_TO_LREAL(count) / gvl.sampleRate /fceLoadTime;
		fbGetPivot(tNow := tr, tTotal := 1.0, pivot => pvt);
		FOR i:=0 TO 5 DO
			FOR j:=0 TO 2 DO
				tipForceDesire[i,j]:=(1-pvt)*tipForceDesireZeros[i,j]+pvt*tipForceDesireGroupB[i,j];
			END_FOR
		END_FOR
	ELSIF count>LREAL_TO_UDINT((tRetract + tWait + tExtend-fceLoadTime)*gvl.sampleRate) AND count<=LREAL_TO_UDINT((tRetract + tWait + tExtend) * gvl.sampleRate) THEN
		tr  := (UDINT_TO_LREAL(count) / gvl.sampleRate-(tRetract + tWait + tExtend-fceLoadTime) )/fceLoadTime;
		fbGetPivot(tNow := tr, tTotal := 1.0, pivot => pvt);
		FOR i:=0 TO 5 BY 2 DO
			FOR j:=0 TO 2 DO
				//tipForceDesire[i,j]:=(1-pvt)*tipForceDesireZeros[i,j]+pvt*tipForceDesireGroupA[i,j];//group A add load
				tipForceDesire[i+1,j]:=(1-pvt)*tipForceDesireGroupB[i+1,j]+pvt*tipForceDesireZeros[i+1,j];//group B reduce load
			END_FOR
		END_FOR
	ELSE
		tipForceDesire:=tipForceDesireGroupB;
	END_IF
//************************************************************************************
	
	IF count < tRetract * gvl.sampleRate THEN
		tTotal := tRetract;
		tNow   := UDINT_TO_LREAL(count) * 1.0 / DINT_TO_LREAL(gvl.sampleRate);
		//jntPosBegin REF= jntAngStart;
		jntPosBegin := jntAngStart;
		FOR i:=0 TO 5 BY 2 DO
			FOR j:=0 TO 2 DO
				jntPosEnd[i,j]:=jntAngRetract[i,j];
				jntPosEnd[i+1,j]:=jntAngStart[i+1,j];
			END_FOR
		END_FOR
	ELSIF count < (tRetract + tWait) * gvl.sampleRate THEN
		tTotal := tWait;
		tNow   := UDINT_TO_LREAL(count) * 1.0 / DINT_TO_LREAL(gvl.sampleRate) - tRetract;
		FOR i:=0 TO 5 BY 2 DO
			FOR j:=0 TO 2 DO
				jntPosBegin[i,j]:=jntAngRetract[i,j];
				jntPosBegin[i+1,j]:=jntAngStart[i+1,j];
				jntPosEnd[i,j]:=jntAngRetract[i,j];
				jntPosEnd[i+1,j]:=jntAngStart[i+1,j];
			END_FOR
		END_FOR
	ELSE 
		tTotal := tExtend;
		tNow   := UDINT_TO_LREAL(count) * 1.0 / DINT_TO_LREAL(gvl.sampleRate) - tRetract - tWait;
		FOR i:=0 TO 5 BY 2 DO
			FOR j:=0 TO 2 DO
				jntPosBegin[i,j]:=jntAngRetract[i,j];
				jntPosBegin[i+1,j]:=jntAngStart[i+1,j];
				jntPosEnd[i,j]:=jntAngExtend[i,j];
				jntPosEnd[i+1,j]:=jntAngStart[i+1,j];
			END_FOR
		END_FOR	
	END_IF	
ELSIF count<=2*(tRetract + tWait + tExtend) * gvl.sampleRate  THEN //leg 1-3-5 recovery

//******************************force compensator******************************
	IF count>LREAL_TO_UDINT((tRetract + tWait + tExtend)*gvl.sampleRate) AND count<=LREAL_TO_UDINT((tRetract + tWait + tExtend+fceLoadTime)* gvl.sampleRate) THEN
		tr  := (UDINT_TO_LREAL(count) / gvl.sampleRate-(tRetract + tWait + tExtend) )/fceLoadTime;
		fbGetPivot(tNow := tr, tTotal := 1.0, pivot => pvt);
		FOR i:=0 TO 5 BY 2 DO
			FOR j:=0 TO 2 DO
				tipForceDesire[i,j]:=(1-pvt)*tipForceDesireZeros[i,j]+pvt*tipForceDesireGroupA[i,j];//group A add load
				tipForceDesire[i+1,j]:=tipForceDesireZeros[i+1,j];//group B zeros load
			END_FOR
		END_FOR		
	ELSIF count>LREAL_TO_UDINT((2*(tRetract + tWait + tExtend)-fceLoadTime)*gvl.sampleRate) AND count<=LREAL_TO_UDINT(2*(tRetract + tWait + tExtend) * gvl.sampleRate) THEN
		tr  := (UDINT_TO_LREAL(count) / gvl.sampleRate-(2*(tRetract + tWait + tExtend)-fceLoadTime) )/fceLoadTime;
		fbGetPivot(tNow := tr, tTotal := 1.0, pivot => pvt);
		FOR i:=0 TO 5 BY 2 DO
			FOR j:=0 TO 2 DO
				tipForceDesire[i,j]:=(1-pvt)*tipForceDesireGroupA[i,j]+pvt*tipForceDesireZeros[i,j];//group A reduce load
				tipForceDesire[i+1,j]:=tipForceDesireZeros[i+1,j];//group B zeros load
			END_FOR
		END_FOR		
	ELSE	
		tipForceDesire:=tipForceDesireGroupA;
	END_IF
//*********************************************************************************
	
	IF count<=(2*tRetract + tWait + tExtend) * gvl.sampleRate THEN
		tTotal := tRetract;
		tNow   := UDINT_TO_LREAL(count) * 1.0 / DINT_TO_LREAL(gvl.sampleRate)-(tRetract + tWait + tExtend);
		FOR i:=0 TO 5 BY 2 DO
			FOR j:=0 TO 2 DO
				jntPosBegin[i,j]:=jntAngExtend[i,j];
				jntPosBegin[i+1,j]:=jntAngStart[i+1,j];
				jntPosEnd[i,j]:=jntAngExtend[i,j];
				jntPosEnd[i+1,j]:=jntAngRetract[i+1,j];
			END_FOR
		END_FOR			
	ELSIF count<=(2*tRetract + 2*tWait + tExtend) * gvl.sampleRate THEN
		tTotal := tWait;
		tNow   := UDINT_TO_LREAL(count) * 1.0 / DINT_TO_LREAL(gvl.sampleRate) - (2*tRetract + tWait + tExtend);
		FOR i:=0 TO 5 BY 2 DO
			FOR j:=0 TO 2 DO
				jntPosBegin[i,j]:=jntAngExtend[i,j];
				jntPosBegin[i+1,j]:=jntAngRetract[i+1,j];
				jntPosEnd[i,j]:=jntAngExtend[i,j];
				jntPosEnd[i+1,j]:=jntAngRetract[i+1,j];
			END_FOR
		END_FOR			
	ELSE
		tTotal := tExtend;
		tNow   := UDINT_TO_LREAL(count) * 1.0 / DINT_TO_LREAL(gvl.sampleRate) - (2*tRetract + 2*tWait + tExtend);
		FOR i:=0 TO 5 BY 2 DO
			FOR j:=0 TO 2 DO
				jntPosBegin[i,j]:=jntAngExtend[i,j];
				jntPosBegin[i+1,j]:=jntAngRetract[i+1,j];
				jntPosEnd[i,j]:=jntAngExtend[i,j];
				jntPosEnd[i+1,j]:=jntAngExtend[i+1,j];
			END_FOR
		END_FOR			
	END_IF
ELSE
	tTotal := 100;
	tNow   := UDINT_TO_LREAL(count) * 1.0 / DINT_TO_LREAL(gvl.sampleRate) - 2*tRetract - 2*tWait - 2*tExtend;
	jntPosBegin :=jntAngExtend;
	jntPosEnd :=jntAngExtend;
	tipForceDesire:=tipForceDesireZeros;
END_IF

getPivot(tNow := tNow, tTotal := tTotal, pivot => pivot, pivotDot => pivotDot);

tipForceDesire:=tipForceDesireZeros;//力补偿control button******************************************************************************************************	
FOR i:=0 TO 5 DO
	tempTipForce[0]:=tipForceDesire[i,0];tempTipForce[1]:=tipForceDesire[i,1];tempTipForce[2]:=tipForceDesire[i,2];
	temJntActPos[0]:=gvl.jntActualPos[i,0];temJntActPos[1]:=gvl.jntActualPos[i,1];temJntActPos[2]:=gvl.jntActualPos[i,2];
	gvl.legCtrl[i].DesireDriveForce(fTipDes:=tempTipForce , motorAng:=temJntActPos , legIndex:=i , fDrvDes=>tempDesJntTrq );
	jntTrqDesire[i,0]:=tempDesJntTrq[0];jntTrqDesire[i,1]:=tempDesJntTrq[1];jntTrqDesire[i,2]:=tempDesJntTrq[2];
END_FOR

FOR i := 0 TO 5 DO
	FOR j := 0 TO 2 DO
		jointPosTarget[i, j] := (1.0 - pivot) * jntPosBegin[i, j] + pivot * jntPosEnd[i, j];
		gvl.jntRefPosLastPlanning[i,j]:=jointPosTarget[i, j] ;
		jointVelTarget[i, j] := - pivotDot * jntPosBegin[i, j] + pivotDot * jntPosEnd[i, j];
		jointFceTarget[i, j] := jntTrqDesire[i,j];
	END_FOR
END_FOR
	
// exit condition
IF count >= (2*tExtend + 2*tRetract + 2*tWait) * gvl.sampleRate + 3 THEN
	isFinished := TRUE;
END_IF
END_METHOD

END_FUNCTION_BLOCK

// ---- POUs/tools/GetPivot.TcPOU
FUNCTION_BLOCK GetPivot
VAR_INPUT
	tNow : LREAL;
	tTotal : LREAL;
END_VAR
VAR_OUTPUT
	pivot : LREAL;
	pivotDot : LREAL;
END_VAR
VAR
	tr : LREAL;
END_VAR

//yk  归一化规划，前半段时间匀加速到0.5，后半段时间匀减速到1
tr := tNow / tTotal;

IF tr <= 0 THEN
	pivot := 0;
	pivotDot := 0;
ELSIF tr <= 0.5 THEN
	pivot := 2.0 * tr * tr;
	pivotDot := 4.0 * tr;
ELSIF tr <= 1 THEN
	pivot := -2.0 * tr * tr + 4.0 * tr - 1.0;
	pivotDot := -4.0 * tr + 4.0;
ELSE
	pivot := 1;
	pivotDot := 0;
END_IF

END_FUNCTION_BLOCK

// ---- POUs/tools/MinDistanceValue.TcPOU
FUNCTION MinDistanceValue : lreal
VAR_INPUT
	rowValue:LREAL;
	refValue:LREAL;
END_VAR
VAR
	rowValueAdd2Pi:LREAL;
	rowValueReduce2Pi:LREAL;
	distance:LREAL;
END_VAR

rowValueAdd2Pi:=rowValue+2*pi;
rowValueReduce2Pi:=rowValue-2*pi;
distance:=Min3Value(ABS(rowValue-refValue),ABS(rowValueAdd2Pi-refValue),ABS(rowValueReduce2Pi-refValue));
IF distance=ABS(rowValue-refValue) THEN
	MinDistanceValue:=rowValue;
ELSIF distance=ABS(rowValueAdd2Pi-refValue) THEN
	MinDistanceValue:=rowValueAdd2Pi;
ELSE
	MinDistanceValue:=rowValueReduce2Pi;
END_IF

END_FUNCTION

// ---- POUs/tools/Min3Value.TcPOU
FUNCTION Min3Value : lreal
VAR_INPUT
	a0:LREAL;
	a1:LREAL;
	a2:LREAL;
END_VAR
VAR
	b: LREAL;
END_VAR

b:=MIN(a0,a1);
IF b<a2 THEN
	 Min3Value:=b;
ELSE
	 Min3Value:=a2;
END_IF

END_FUNCTION

// ---- POUs/GaitPlanner/StaticWalkGait.TcPOU
FUNCTION_BLOCK StaticWalkGait
VAR_INPUT
END_VAR
VAR_OUTPUT
END_VAR
VAR
	//input
	H:LREAL :=0.09;//step height
	L:LREAL :=0.1;//step length
	La:lreal :=0;// lateral step length
	period:LREAL:=2;
	
	N:INT :=1;//total steps  number
	Yaw:LREAL :=0;// total Yaw angle (unit:degree)
	
	//intermediate variable
	quit_flag  : BOOL;
	require_stop_flag:BOOL;
	start_flag:BOOL;
	BodyHeight:LREAL;//body height
	SampleRate :UDINT :=1000;
	totalcount:DINT :=TRUNC(period*SampleRate);//duration time of half step
	delta_t:LREAL :=1.0/SampleRate;//sample time
	dYaw:LREAL :=Yaw/(2.0*N);// rotation angle in every half step
	gait_cycle   : UDINT := 0;//count time from select this step
	period_count :UDINT := 0;
	SupportLegA:INT :=1;// legs of group A are supporting and ones of group B are swing
	SupportLegB:INT :=2;// legs of group B are supporting and ones of group A are swing
	SupportLegAB:INT :=3;// legs of group A and B are supporting 
	SupportPhase:INT;
		// trajectory planning
	joint_ref_pos_init : ARRAY[0..5] OF Vec3;
	joint_ref_pos_target : ARRAY[0..5] OF Vec3;
	
	body_ref_pos_init : Vec3;
	body_ref_pos_target : Vec3;
	body_ref_ang_init : Vec3;
	body_ref_ang_target : Vec3;
    leg_ref_pos_init : ARRAY[0..5] OF Vec3;
	jointPosLast   : ARRAY[0..5, 0..2] OF LREAL; 
	leg_ref_pos_target:ARRAY[0..5] OF Vec3;
	leg_ref_pos_init_wrt_hip : ARRAY[0..5] OF Vec3;
	leg_ref_pos_target_wrt_hip : ARRAY[0..5] OF Vec3;

	body_ref_pos : Vec3;
	body_ref_ang : Vec3;
	body_ref_vel:vec3;
	body_ref_angvel:vec3;
	
    leg_ref_pos : ARRAY[0..5] OF Vec3;
	leg_ref_pos_wrt_hip : ARRAY[0..5] OF Vec3;
	
	body_ref_pos_next : Vec3;
	body_ref_ang_next : Vec3;
    leg_ref_pos_next : ARRAY[0..5] OF Vec3;
	leg_ref_pos_next_wrt_hip : ARRAY[0..5] OF Vec3;
	leg_ref_vel_next_wrt_hip : ARRAY[0..5] OF Vec3;
	
	jointPosTarget  : ARRAY[0..5, 0..2] OF LREAL; 
	jointVelTarget  : ARRAY[0..5, 0..2] OF LREAL;  
	jointFceTarget  : ARRAY[0..5, 0..2] OF LREAL;  
	
	fbRotmat : RotM;
	Rb : Mat3;
	hip_pos_j  : Vec3;
	leg_pos_wrt_com : Vec3;
	Rleg : ARRAY[0..5] OF Mat3;
	Rb_actual : Mat3;
	tip_actual_pos_wrt_world : ARRAY[0..5] OF Vec3;
	
	// robot paramates
	hip_pos : ARRAY[0..5, 0..2] OF LREAL := [-0.369,  -0.125, 0,
                                             0,  -0.28, 0,
                                             0.36, -0.125, 0,
                                             0.36, 0.125, 0,
											 0,0.28,0,
											 -0.369,0.125,0];
	
	//outpot
	isFinished      : BOOL := FALSE;
		
	leg_index_mapping : ARRAY[0..5] OF INT := [1, 2, 3, 4,5,6];
			// output test
	joint_ref_pos   : ARRAY[0..5] OF Vec3;
	joint_ref_vel   : ARRAY[0..5] OF Vec3;
	joint_ref_fce   : ARRAY[0..5] OF Vec3; 
	hip_ref_pos_init: ARRAY[0..5] OF vec3;
	
	joint_ref_pos_last : ARRAY[0..5] OF Vec3;
	joint_ref_vel_diff : ARRAY[0..5] OF Vec3;
	Rb_target1 : Mat3;
	Rb_target2 : Mat3;
	hip_ref_pos_rot: ARRAY[0..5] OF vec3;
	leg_ref_pos_rot:ARRAY[0..5] OF vec3;
	leg_ref_pos_wrt_body:ARRAY[0..5] OF vec3;
END_VAR

METHOD BodyStabilize : BOOL
VAR_INPUT
END_VAR
END_METHOD

METHOD DoPlanning : BOOL
VAR_INPUT
	count: UDINT;
END_VAR

VAR
	i: INT;
	j: INT;
END_VAR
IF count = 0 THEN
	isFinished := FALSE;
	Initialize();
	totalcount :=TRUNC(period*SampleRate);//duration time of half step
	dYaw:=Yaw/(2.0*N)*pi/180;
	IF Yaw=0 THEN
		La:=La;
	ELSE
		La:=0;
	END_IF
END_IF
StateMachine();
BodyStabilize();
TrjPlanning();

// count
gait_cycle := gait_cycle + 1;
IF require_stop_flag=TRUE THEN
	isFinished := TRUE;
	quit_flag := FALSE;
	gait_cycle:=0;
	// link to physical outputs
	FOR i := 0 TO 5 DO
		FOR j := 0 TO 2 DO
			jointPosTarget[i, j] := joint_ref_pos[i].data[j];
			jointVelTarget[i, j] := 0;
			jointFceTarget[i, j] := 0;
		END_FOR
	END_FOR
END_IF

IF quit_flag AND SupportPhase = SupportLegAB THEN
	isFinished := TRUE;
	quit_flag := FALSE;
	gait_cycle:=0;
END_IF
END_METHOD

METHOD Initialize : BOOL
VAR_INPUT
END_VAR
VAR
	i, j : INT;
	sum_height : LREAL := 0;
	leg_pos    : ARRAY[0..2] OF LREAL;
END_VAR
Rleg[0]:=SetMat3(1,0,0,0,0,-1,0,1,0);
Rleg[1]:=SetMat3(-1,0,0,0,0,1,0,1,0,);
Rleg[2]:=SetMat3(-1,0,0,0,0,1,0,1,0);
Rleg[3]:=SetMat3(-1,0,0,0,0,1,0,1,0);
Rleg[4]:=SetMat3( -1,0,0,0,0,1,0,1,0);
Rleg[5]:=SetMat3(1,0,0,0,0,-1,0,1,0);

SupportPhase:=SupportLegAB;
quit_flag :=FALSE;
require_stop_flag:=false;
gait_cycle := 0;

// init trajectory
FOR i := 0 TO 5 DO
	FOR j := 0 TO 2 DO
		IF ABS(gvl.jntLastRefPos[i, j] - gvl.jntActualPos[i, j]) < gvl.walk_threshold_value THEN//gvl.jntLastRefPos上次规划值，或者力控开始时的值
			joint_ref_pos_init[i].data[j] := gvl.jntLastRefPos[i, j];
		ELSE
			joint_ref_pos_init[i].data[j] := gvl.jntActualPos[i, j];
		END_IF
		jointPosLast[i,j]:=joint_ref_pos_init[i].data[j];
	END_FOR
END_FOR

sum_height := 0;
FOR j := 0 TO 5 DO
	// FK
	gvl.legCtrl[j].ForwardKinetics(motorAngles := joint_ref_pos_init[j].data,legIndex:=j, tipPosition => leg_pos);
	leg_ref_pos_init_wrt_hip[j] := SetVec3(leg_pos[0], leg_pos[1], leg_pos[2]);
	sum_height := sum_height + (-leg_ref_pos_init_wrt_hip[j].data[1]);
END_FOR
body_ref_pos_init := SetVec3(0, 0, sum_height/6.0);
body_ref_ang_init := SetVec3(gvl.rpy_model[0], gvl.rpy_model[1], 0);                            

fbRotMat(yaw := 0, 
	     pitch := gvl.rpy_model[1],
		 roll := gvl.rpy_model[0],
		 rm => Rb_actual);
FOR j:=0 TO 5 DO
		hip_pos_j := SetVec3(hip_pos[j, 0], hip_pos[j, 1], hip_pos[j, 2]);
		hip_ref_pos_init[j]:=VecAdd(MatMulVec(Rb_actual,hip_pos_j ),body_ref_pos_init);	
END_FOR
FOR j := 0 TO 5 DO
	hip_pos_j := SetVec3(hip_pos[j, 0], hip_pos[j, 1], hip_pos[j, 2]);
	leg_pos_wrt_com := VecAdd(MatMulVec(Rleg[j], leg_ref_pos_init_wrt_hip[j]), hip_pos_j);
    leg_ref_pos_init[j] := VecAdd(body_ref_pos_init, MatMulVec(Rb_actual, leg_pos_wrt_com));
END_FOR

body_ref_pos := body_ref_pos_init;
body_ref_ang := body_ref_ang_init;
leg_ref_pos := leg_ref_pos_init;
leg_ref_pos_wrt_hip := leg_ref_pos_init_wrt_hip;

FOR i := 0 TO 5 DO
	FOR j := 0 TO 2 DO
		jointPosTarget[i, j] := joint_ref_pos_init[i].data[j];
		jointVelTarget[i, j] := 0;
		jointFceTarget[i, j] := 0;
	END_FOR
END_FOR
END_METHOD

METHOD StateMachine : BOOL
VAR_INPUT
END_VAR
period_count:=gait_cycle MOD totalcount;
 
IF gait_cycle/totalcount = 0 THEN
	SupportPhase:=SupportLegA;
ELSIF gait_cycle/totalcount=2*N-1 THEN
	SupportPhase:=SupportLegB;
ELSIF (gait_cycle/totalcount MOD 2)=1 THEN
	SupportPhase:=SupportLegB;
ELSE
	SupportPhase:=SupportLegA;
END_IF
IF gait_cycle>=2*N*totalcount THEN
	SupportPhase:=SupportLegAB;
	quit_flag:=TRUE;
END_IF
END_METHOD

METHOD TrjPlanning : BOOL
VAR_INPUT
END_VAR

VAR
	i: INT;
	j: INT;
	temp :vec3;
	temp1: Vec3;
	temp2: Vec3;
	temp3: Vec3;
	tmp:vec3;
	tip_pos, tip_vel : Vec3;
	fbElipseInterpolation:ElipseInterpolation;
	fbHermitInterpolation:HermitInterpolation;
	body_ref_vel_init: Vec3;
	body_ref_angvel_init:vec3;
	body_ref_vel_target: Vec3;
	body_ref_angvel_target:vec3;
	leg_ref_pos_wrt_com_j : Vec3;
	stopflag: BOOL;
	
	jointTmpPosLast: ARRAY[0..2] OF LREAL;
END_VAR
IF gait_cycle/totalcount = 0 THEN
	//the first step
	//update target toe position 
	FOR i:=0 TO 5  BY 2 DO //0-2-4 support
		FOR j:=0 TO 2  DO
			leg_ref_pos_target[i].data[j]:=leg_ref_pos_init[i].data[j];
		END_FOR
	END_FOR
	temp:=SetVec3(L/2*COS(dYaw),L/2*SIN(dYaw)+La/2,0);
	fbRotMat(yaw := 2*dYaw, pitch := 0, roll := 0, rm => Rb_target2);
	fbRotMat(yaw := 0, pitch := 0,roll := 0,rm => Rb_target1);
	FOR j:=0 TO 5 DO
		leg_ref_pos_wrt_body[j]:= MatMulVec( MatTranspose(Rb_target1), VecAdd(leg_ref_pos_init[j],VecNeg(body_ref_pos_init)));
		leg_ref_pos_rot[j]:=VecAdd( MatMulVec(Rb_target2,leg_ref_pos_wrt_body[j] ),VecNeg(MatMulVec(Rb_target1,leg_ref_pos_wrt_body[j])));
	END_FOR
		 
	FOR i:=1 TO 5 BY 2 DO //1-3-5 swing
		FOR j:=0 TO 1  DO
			leg_ref_pos_target[i].data[j]:=leg_ref_pos_init[i].data[j]+temp.data[j]+leg_ref_pos_rot[i].data[j];
		END_FOR
		leg_ref_pos_target[i].data[2]:=leg_ref_pos_init[i].data[2]+temp.data[2];
	END_FOR
	//update body target position
	temp1:=SetVec3(L/4*COS(dYaw),L/4*SIN(dYaw)+La/4,0);
	temp2:=SetVec3(0,0,dYaw);
	FOR i:=0 TO 2 DO
		body_ref_pos_target.data[i]:=body_ref_pos_init.data[i]+temp1.data[i];
		body_ref_ang_target.data[i]:=body_ref_ang_init.data[i]+temp2.data[i];
	END_FOR
	//update body velocity
	body_ref_vel_init:=setvec3(0,0,0);
	body_ref_angvel_init:=setvec3(0,0,0);
	body_ref_vel_target:=setvec3(0.5*L/(totalcount*delta_t)*COS(dYaw),0.5*L/(totalcount*delta_t)*SIN(dYaw)+0.5*La/(totalcount*delta_t),0);
	body_ref_angvel_target:=setvec3(0,0,dYaw/(totalcount*delta_t));
	// planing toe trajectory
	FOR i:=0 TO 5 BY 2 DO//0-2-4 support
		FOR j:=0 TO 2 DO 
			leg_ref_pos[i].data[j]:=leg_ref_pos_init[i].data[j];
		END_FOR
	END_FOR
	FOR i:=1 TO 5 BY 2 DO//1-3-5 swing
		fbElipseInterpolation(x0:=leg_ref_pos_init[i].data[0] , y0:=leg_ref_pos_init[i].data[1] , z0:=leg_ref_pos_init[i].data[2] , x1:=leg_ref_pos_target[i].data[0] , 
		y1:=leg_ref_pos_target[i].data[1] , z1:=leg_ref_pos_target[i].data[2] , h:=H , T:=totalcount*delta_t , t0:=0 , tNow:= period_count*delta_t, 
		x=>leg_ref_pos[i].data[0] , y=>leg_ref_pos[i].data[1] , z=>leg_ref_pos[i].data[2] );
	END_FOR
	// planing body trajectory
	FOR i:=0 TO 2 DO
		fbHermitInterpolation(t0:=0 , T:=totalcount*delta_t , y0:=body_ref_pos_init.data[i] , y1:=body_ref_pos_target.data[i] , v0:=body_ref_vel_init.data[i] , 
		v1:=body_ref_vel_target.data[i] , tNow:=period_count*delta_t , y=>body_ref_pos.data[i] , v=> body_ref_vel.data[i]);
		fbHermitInterpolation(t0:=0 , T:=totalcount*delta_t , y0:=body_ref_ang_init.data[i] , y1:=body_ref_ang_target.data[i] , v0:=body_ref_angvel_init.data[i] , 
		v1:=body_ref_angvel_target.data[i] , tNow:=period_count*delta_t , y=>body_ref_ang.data[i] , v=> body_ref_angvel.data[i]);		
	END_FOR
	
ELSIF gait_cycle/totalcount= 2*N-1 THEN
	//the last step
	IF period_count=0 THEN
		leg_ref_pos_init:=leg_ref_pos_target;
		body_ref_pos_init:=body_ref_pos_target;
		body_ref_ang_init:=body_ref_ang_target;
	END_IF
	//update target toe position 
	temp:=SetVec3(L/2*COS(dYaw),L/2*SIN(dYaw)+La/2,0);
	fbRotMat(yaw := 2*dYaw, pitch := 0,roll := 0,rm => Rb_target2);
	fbRotMat(yaw := 0, pitch := 0,roll := 0,rm => Rb_target1);
	FOR j:=0 TO 5 DO
		leg_ref_pos_wrt_body[j]:= MatMulVec( MatTranspose(Rb_target1), VecAdd(leg_ref_pos_init[j],VecNeg(body_ref_pos_init)));
		leg_ref_pos_rot[j]:=VecAdd( MatMulVec(Rb_target2,leg_ref_pos_wrt_body[j] ),VecNeg(MatMulVec(Rb_target1,leg_ref_pos_wrt_body[j])));	
	END_FOR
	FOR i:=0 TO 5  BY 2 DO //0-2-4 swing target position
		FOR j:=0 TO 2  DO
			leg_ref_pos_target[i].data[j]:=leg_ref_pos_init[i].data[j]+temp.data[j]+leg_ref_pos_rot[i].data[j];
		END_FOR
	END_FOR
	
